LIN {X 0,Y 313.371,Z 298.457,A -85,B 0,C 180,E1 -15702.885,E2 -15702.885} C_VEL
LIN {X 0,Y 315.381,Z 300.73,A -85,B 0,C 180,E1 -15703.354,E2 -15703.354} C_VEL
LIN {X 0,Y 318.068,Z 304.811,A -85,B 0,C 180,E1 -15703.999,E2 -15703.999} C_VEL
LIN {X 0,Y 319.431,Z 306.632,A -85,B 0,C 180,E1 -15704.311,E2 -15704.311} C_VEL
LIN {X 0,Y 325.646,Z 315.457,A -85,B 0,C 180,E1 -15705.697,E2 -15705.697} C_VEL
LIN {X 0,Y 333.8,Z 327.772,A -85,B 0,C 180,E1 -15707.413,E2 -15707.413} C_VEL
LIN {X 0,Y 340.468,Z 338.749,A -85,B 0,C 180,E1 -15708.748,E2 -15708.748} C_VEL
LIN {X 0,Y 347.31,Z 351.998,A -85,B 0,C 180,E1 -15710.09,E2 -15710.09} C_VEL
LIN {X 0,Y 349.125,Z 355.68,A -85,B 0,C 180,E1 -15710.437,E2 -15710.437} C_VEL
LIN {X 0,Y 343.663,Z 493.802,A -85,B 0,C 180,E1 -15713.33,E2 -15713.33} C_VEL
LIN {X 0,Y 342.311,Z 510.914,A -85,B 0,C 180,E1 -15713.87,E2 -15713.87} C_VEL
LIN {X 0,Y 340.606,Z 527.054,A -85,B 0,C 180,E1 -15714.618,E2 -15714.618} C_VEL
LIN {X 0,Y 338.492,Z 542.365,A -85,B 0,C 180,E1 -15715.544,E2 -15715.544} C_VEL
LIN {X 0,Y 335.932,Z 557.671,A -85,B 0,C 180,E1 -15716.726,E2 -15716.726} C_VEL
LIN {X 0,Y 333.332,Z 571.386,A -85,B 0,C 180,E1 -15718.039,E2 -15718.039} C_VEL
LIN {X 0,Y 330.539,Z 584.215,A -85,B 0,C 180,E1 -15719.494,E2 -15719.494} C_VEL
LIN {X 0,Y 327.433,Z 597.477,A -85,B 0,C 180,E1 -15721.298,E2 -15721.298} C_VEL
LIN {X 0,Y 324.398,Z 609.578,A -85,B 0,C 180,E1 -15723.286,E2 -15723.286} C_VEL
LIN {X 0,Y 321.492,Z 620.685,A -85,B 0,C 180,E1 -15725.459,E2 -15725.459} C_VEL
LIN {X 0,Y 318.88,Z 630.612,A -85,B 0,C 180,E1 -15727.769,E2 -15727.769} C_VEL
LIN {X 0,Y 316.636,Z 639.434,A -85,B 0,C 180,E1 -15730.215,E2 -15730.215} C_VEL
LIN {X 0,Y 314.486,Z 647.965,A -85,B 0,C 180,E1 -15733.111,E2 -15733.111} C_VEL
LIN {X 0,Y 312.79,Z 655.524,A -85,B 0,C 180,E1 -15736.354,E2 -15736.354} C_VEL
LIN {X 0,Y 311.681,Z 661.259,A -85,B 0,C 180,E1 -15739.608,E2 -15739.608} C_VEL
LIN {X 0,Y 311.176,Z 664.614,A -85,B 0,C 180,E1 -15742.212,E2 -15742.212} C_VEL
LIN {X 0,Y 310.877,Z 667.053,A -85,B 0,C 180,E1 -15744.812,E2 -15744.812} C_VEL
LIN {X 0,Y 310.734,Z 668.437,A -85,B 0,C 180,E1 -15747.407,E2 -15747.407} C_VEL
LIN {X 0,Y 310.695,Z 668.97,A -85,B 0,C 180,E1 -15750,E2 -15750} C_VEL
LIN {X 0,Y 310.734,Z 668.477,A -85,B 0,C 180,E1 -15752.593,E2 -15752.593} C_VEL
LIN {X 0,Y 310.876,Z 667.132,A -85,B 0,C 180,E1 -15755.188,E2 -15755.188} C_VEL
LIN {X 0,Y 311.171,Z 664.734,A -85,B 0,C 180,E1 -15757.788,E2 -15757.788} C_VEL
LIN {X 0,Y 311.656,Z 661.427,A -85,B 0,C 180,E1 -15760.393,E2 -15760.393} C_VEL
LIN {X 0,Y 312.759,Z 655.741,A -85,B 0,C 180,E1 -15763.647,E2 -15763.647} C_VEL
LIN {X 0,Y 314.454,Z 648.254,A -85,B 0,C 180,E1 -15766.891,E2 -15766.891} C_VEL
LIN {X 0,Y 316.57,Z 639.766,A -85,B 0,C 180,E1 -15769.789,E2 -15769.789} C_VEL
LIN {X 0,Y 318.736,Z 631.273,A -85,B 0,C 180,E1 -15772.167,E2 -15772.167} C_VEL
LIN {X 0,Y 321.437,Z 621.161,A -85,B 0,C 180,E1 -15774.546,E2 -15774.546} C_VEL
LIN {X 0,Y 324.293,Z 610.151,A -85,B 0,C 180,E1 -15776.723,E2 -15776.723} C_VEL
LIN {X 0,Y 327.588,Z 597.113,A -85,B 0,C 180,E1 -15778.862,E2 -15778.862} C_VEL
LIN {X 0,Y 330.674,Z 583.796,A -85,B 0,C 180,E1 -15780.669,E2 -15780.669} C_VEL
LIN {X 0,Y 333.621,Z 570.298,A -85,B 0,C 180,E1 -15782.18,E2 -15782.18} C_VEL
LIN {X 0,Y 336.173,Z 556.682,A -85,B 0,C 180,E1 -15783.462,E2 -15783.462} C_VEL
LIN {X 0,Y 338.696,Z 541.625,A -85,B 0,C 180,E1 -15784.613,E2 -15784.613} C_VEL
LIN {X 0,Y 339.449,Z 536.57,A -85,B 0,C 180,E1 -15784.931,E2 -15784.931} C_VEL
LIN {X 0,Y 339.734,Z 531.151,A -85,B 0,C 180,E1 -15785.32,E2 -15785.32} C_VEL
LIN {X 0,Y 337.206,Z 513.489,A -85,B 0,C 180,E1 -15786.764,E2 -15786.764} C_VEL
LIN {X 0,Y 337.05,Z 507.877,A -85,B 0,C 180,E1 -15787.068,E2 -15787.068} C_VEL
LIN {X 0,Y 338.19,Z 491.988,A -85,B 0,C 180,E1 -15787.544,E2 -15787.544} C_VEL
LIN {X 0,Y 343.655,Z 358.179,A -85,B 0,C 180,E1 -15790.378,E2 -15790.378} C_VEL
LIN {X 0,Y 336.006,Z 343.116,A -85,B 0,C 180,E1 -15791.927,E2 -15791.927} C_VEL
LIN {X 0,Y 327.751,Z 329.585,A -85,B 0,C 180,E1 -15793.647,E2 -15793.647} C_VEL
LIN {X 0,Y 317.849,Z 314.862,A -85,B 0,C 180,E1 -15795.853,E2 -15795.853} C_VEL
LIN {X 0,Y 312.292,Z 307.072,A -85,B 0,C 180,E1 -15797.179,E2 -15797.179} C_VEL
LIN {X 0,Y 309.294,Z 303.031,A -85,B 0,C 180,E1 -15797.923,E2 -15797.923} C_VEL
LIN {X 0,Y 308.538,Z 301.775,A -85,B 0,C 180,E1 -15798.123,E2 -15798.123} C_VEL
LIN {X 0,Y 306.51,Z 299.73,A -85,B 0,C 180,E1 -15798.621,E2 -15798.621} C_VEL
LIN {X 0,Y 305.504,Z 297.232,A -85,B 0,C 180,E1 -15798.925,E2 -15798.925} C_VEL
LIN {X 0,Y 305.437,Z 296.736,A -85,B 0,C 180,E1 -15798.999,E2 -15798.999} C_VEL
LIN {X 0,Y 305.474,Z 296.741,A -85,B 0,C 180,E1 -15801.597,E2 -15801.597} C_VEL
LIN {X 0,Y 305.461,Z 296.748,A -85,B 0,C 180,E1 -15804.886,E2 -15804.886} C_VEL
LIN {X 0,Y 305.448,Z 296.735,A -85,B 0,C 180,E1 -15808.355,E2 -15808.355} C_VEL
LIN {X 0,Y 305.511,Z 296.727,A -85,B 0,C 180,E1 -15811.113,E2 -15811.113} C_VEL
LIN {X 0,Y 305.569,Z 296.727,A -85,B 0,C 180,E1 -15814.088,E2 -15814.088} C_VEL
LIN {X 0,Y 305.498,Z 296.717,A -85,B 0,C 180,E1 -15818.403,E2 -15818.403} C_VEL
LIN {X 0,Y 305.588,Z 296.732,A -85,B 0,C 180,E1 -15821.217,E2 -15821.217} C_VEL
LIN {X 0,Y 305.647,Z 296.704,A -85,B 0,C 180,E1 -15825.349,E2 -15825.349} C_VEL
LIN {X 0,Y 305.636,Z 296.7,A -85,B 0,C 180,E1 -15829.399,E2 -15829.399} C_VEL
LIN {X 0,Y 305.811,Z 296.687,A -85,B 0,C 180,E1 -15832.074,E2 -15832.074} C_VEL
LIN {X 0,Y 305.687,Z 296.715,A -85,B 0,C 180,E1 -15834.723,E2 -15834.723} C_VEL
LIN {X 0,Y 305.955,Z 296.666,A -85,B 0,C 180,E1 -15838.684,E2 -15838.684} C_VEL
LIN {X 0,Y 305.955,Z 296.683,A -85,B 0,C 180,E1 -15841.316,E2 -15841.316} C_VEL
LIN {X 0,Y 305.85,Z 296.696,A -85,B 0,C 180,E1 -15846.597,E2 -15846.597} C_VEL
LIN {X 0,Y 305.734,Z 296.693,A -85,B 0,C 180,E1 -15849.26,E2 -15849.26} C_VEL
LIN {X 0,Y 305.587,Z 296.732,A -85,B 0,C 180,E1 -15853.296,E2 -15853.296} C_VEL
LIN {X 0,Y 305.592,Z 296.729,A -85,B 0,C 180,E1 -15856.02,E2 -15856.02} C_VEL
LIN {X 0,Y 305.575,Z 296.736,A -85,B 0,C 180,E1 -15859.445,E2 -15859.445} C_VEL
LIN {X 0,Y 305.488,Z 296.749,A -85,B 0,C 180,E1 -15863.041,E2 -15863.041} C_VEL
LIN {X 0,Y 305.545,Z 296.743,A -85,B 0,C 180,E1 -15866.227,E2 -15866.227} C_VEL
LIN {X 0,Y 305.494,Z 296.749,A -85,B 0,C 180,E1 -15869.05,E2 -15869.05} C_VEL
LIN {X 0,Y 305.442,Z 296.757,A -85,B 0,C 180,E1 -15871.952,E2 -15871.952} C_VEL
LIN {X 0,Y 305.46,Z 296.75,A -85,B 0,C 180,E1 -15875.113,E2 -15875.113} C_VEL
LIN {X 0,Y 305.447,Z 296.757,A -85,B 0,C 180,E1 -15878.529,E2 -15878.529} C_VEL
LIN {X 0,Y 305.465,Z 296.923,A -85,B 0,C 180,E1 -15879.468,E2 -15879.468} C_VEL
LIN {X 0,Y 308.218,Z 303.518,A -85,B 0,C 180,E1 -15881.505,E2 -15881.505} C_VEL
LIN {X 0,Y 316.88,Z 316.875,A -85,B 0,C 180,E1 -15883.664,E2 -15883.664} C_VEL
LIN {X 0,Y 324.584,Z 329.236,A -85,B 0,C 180,E1 -15885.438,E2 -15885.438} C_VEL
LIN {X 0,Y 332.597,Z 343.649,A -85,B 0,C 180,E1 -15887.189,E2 -15887.189} C_VEL
LIN {X 0,Y 340.914,Z 360.154,A -85,B 0,C 180,E1 -15888.915,E2 -15888.915} C_VEL
LIN {X 0,Y 343.483,Z 365.809,A -85,B 0,C 180,E1 -15889.437,E2 -15889.437} C_VEL
LIN {X 0,Y 337.406,Z 512.132,A -85,B 0,C 180,E1 -15892.54,E2 -15892.54} C_VEL
LIN {X 0,Y 335.817,Z 529.145,A -85,B 0,C 180,E1 -15893.104,E2 -15893.104} C_VEL
LIN {X 0,Y 333.935,Z 544.026,A -85,B 0,C 180,E1 -15893.801,E2 -15893.801} C_VEL
LIN {X 0,Y 331.666,Z 559.189,A -85,B 0,C 180,E1 -15894.731,E2 -15894.731} C_VEL
LIN {X 0,Y 328.916,Z 574.15,A -85,B 0,C 180,E1 -15895.883,E2 -15895.883} C_VEL
LIN {X 0,Y 325.719,Z 589.41,A -85,B 0,C 180,E1 -15897.356,E2 -15897.356} C_VEL
LIN {X 0,Y 322.401,Z 603.395,A -85,B 0,C 180,E1 -15899.003,E2 -15899.003} C_VEL
LIN {X 0,Y 319.483,Z 615.351,A -85,B 0,C 180,E1 -15900.696,E2 -15900.696} C_VEL
LIN {X 0,Y 316.666,Z 626.009,A -85,B 0,C 180,E1 -15902.465,E2 -15902.465} C_VEL
LIN {X 0,Y 313.934,Z 636.294,A -85,B 0,C 180,E1 -15904.473,E2 -15904.473} C_VEL
LIN {X 0,Y 311.298,Z 646.17,A -85,B 0,C 180,E1 -15906.729,E2 -15906.729} C_VEL
LIN {X 0,Y 308.826,Z 655.677,A -85,B 0,C 180,E1 -15909.345,E2 -15909.345} C_VEL
LIN {X 0,Y 306.925,Z 663.639,A -85,B 0,C 180,E1 -15911.994,E2 -15911.994} C_VEL
LIN {X 0,Y 305.507,Z 670.29,A -85,B 0,C 180,E1 -15914.661,E2 -15914.661} C_VEL
LIN {X 0,Y 304.548,Z 675.693,A -85,B 0,C 180,E1 -15917.336,E2 -15917.336} C_VEL
LIN {X 0,Y 304.001,Z 679.031,A -85,B 0,C 180,E1 -15919.342,E2 -15919.342} C_VEL
LIN {X 0,Y 303.684,Z 682.467,A -85,B 0,C 180,E1 -15922.019,E2 -15922.019} C_VEL
LIN {X 0,Y 303.595,Z 684.967,A -85,B 0,C 180,E1 -15924.687,E2 -15924.687} C_VEL
LIN {X 0,Y 303.594,Z 686.378,A -85,B 0,C 180,E1 -15927.346,E2 -15927.346} C_VEL
LIN {X 0,Y 303.601,Z 686.908,A -85,B 0,C 180,E1 -15930,E2 -15930} C_VEL
LIN {X 0,Y 303.594,Z 686.371,A -85,B 0,C 180,E1 -15932.654,E2 -15932.654} C_VEL
LIN {X 0,Y 303.623,Z 684.76,A -85,B 0,C 180,E1 -15935.545,E2 -15935.545} C_VEL
LIN {X 0,Y 303.684,Z 682.446,A -85,B 0,C 180,E1 -15937.982,E2 -15937.982} C_VEL
LIN {X 0,Y 304.001,Z 679.004,A -85,B 0,C 180,E1 -15940.658,E2 -15940.658} C_VEL
LIN {X 0,Y 305.004,Z 673.131,A -85,B 0,C 180,E1 -15944.001,E2 -15944.001} C_VEL
LIN {X 0,Y 306.516,Z 665.413,A -85,B 0,C 180,E1 -15947.342,E2 -15947.342} C_VEL
LIN {X 0,Y 308.603,Z 656.719,A -85,B 0,C 180,E1 -15950.322,E2 -15950.322} C_VEL
LIN {X 0,Y 310.955,Z 647.339,A -85,B 0,C 180,E1 -15952.946,E2 -15952.946} C_VEL
LIN {X 0,Y 313.537,Z 637.697,A -85,B 0,C 180,E1 -15955.207,E2 -15955.207} C_VEL
LIN {X 0,Y 316.215,Z 627.523,A -85,B 0,C 180,E1 -15957.251,E2 -15957.251} C_VEL
LIN {X 0,Y 319.449,Z 615.221,A -85,B 0,C 180,E1 -15959.308,E2 -15959.308} C_VEL
LIN {X 0,Y 322.649,Z 602.059,A -85,B 0,C 180,E1 -15961.153,E2 -15961.153} C_VEL
LIN {X 0,Y 325.761,Z 588.634,A -85,B 0,C 180,E1 -15962.713,E2 -15962.713} C_VEL
LIN {X 0,Y 328.889,Z 573.901,A -85,B 0,C 180,E1 -15964.12,E2 -15964.12} C_VEL
LIN {X 0,Y 331.819,Z 557.903,A -85,B 0,C 180,E1 -15965.344,E2 -15965.344} C_VEL
LIN {X 0,Y 334.109,Z 542.363,A -85,B 0,C 180,E1 -15966.271,E2 -15966.271} C_VEL
LIN {X 0,Y 336.028,Z 526.804,A -85,B 0,C 180,E1 -15966.963,E2 -15966.963} C_VEL
LIN {X 0,Y 337.482,Z 510.229,A -85,B 0,C 180,E1 -15967.484,E2 -15967.484} C_VEL
LIN {X 0,Y 343.385,Z 365.697,A -85,B 0,C 180,E1 -15970.551,E2 -15970.551} C_VEL
LIN {X 0,Y 335.117,Z 348.583,A -85,B 0,C 180,E1 -15972.244,E2 -15972.244} C_VEL
LIN {X 0,Y 326.72,Z 332.985,A -85,B 0,C 180,E1 -15974.048,E2 -15974.048} C_VEL
LIN {X 0,Y 318.181,Z 318.811,A -85,B 0,C 180,E1 -15975.99,E2 -15975.99} C_VEL
LIN {X 0,Y 313.283,Z 311.23,A -85,B 0,C 180,E1 -15977.167,E2 -15977.167} C_VEL
LIN {X 0,Y 308.364,Z 303.718,A -85,B 0,C 180,E1 -15978.411,E2 -15978.411} C_VEL
LIN {X 0,Y 307.25,Z 301.662,A -85,B 0,C 180,E1 -15979.011,E2 -15979.011} C_VEL
LIN {X 0,Y 305.448,Z 296.74,A -85,B 0,C 180,E1 -15980.583,E2 -15980.583} C_VEL
LIN {X 0,Y 305.479,Z 296.742,A -85,B 0,C 180,E1 -15983.632,E2 -15983.632} C_VEL
LIN {X 0,Y 305.463,Z 296.745,A -85,B 0,C 180,E1 -15986.483,E2 -15986.483} C_VEL
LIN {X 0,Y 305.461,Z 296.742,A -85,B 0,C 180,E1 -15989.591,E2 -15989.591} C_VEL
LIN {X 0,Y 305.519,Z 296.735,A -85,B 0,C 180,E1 -15992.609,E2 -15992.609} C_VEL
LIN {X 0,Y 305.506,Z 296.737,A -85,B 0,C 180,E1 -15995.539,E2 -15995.539} C_VEL
LIN {X 0,Y 305.517,Z 296.709,A -85,B 0,C 180,E1 -15999.815,E2 -15999.815} C_VEL
LIN {X 0,Y 305.573,Z 296.732,A -85,B 0,C 180,E1 -16002.603,E2 -16002.603} C_VEL
LIN {X 0,Y 305.647,Z 296.697,A -85,B 0,C 180,E1 -16005.349,E2 -16005.349} C_VEL
LIN {X 0,Y 305.634,Z 296.725,A -85,B 0,C 180,E1 -16009.4,E2 -16009.4} C_VEL
LIN {X 0,Y 305.795,Z 296.681,A -85,B 0,C 180,E1 -16012.074,E2 -16012.074} C_VEL
LIN {X 0,Y 305.685,Z 296.69,A -85,B 0,C 180,E1 -16014.724,E2 -16014.724} C_VEL
LIN {X 0,Y 305.954,Z 296.672,A -85,B 0,C 180,E1 -16018.684,E2 -16018.684} C_VEL
LIN {X 0,Y 305.954,Z 296.649,A -85,B 0,C 180,E1 -16021.316,E2 -16021.316} C_VEL
LIN {X 0,Y 305.686,Z 296.716,A -85,B 0,C 180,E1 -16025.277,E2 -16025.277} C_VEL
LIN {X 0,Y 305.795,Z 296.667,A -85,B 0,C 180,E1 -16027.926,E2 -16027.926} C_VEL
LIN {X 0,Y 305.602,Z 296.73,A -85,B 0,C 180,E1 -16031.945,E2 -16031.945} C_VEL
LIN {X 0,Y 305.636,Z 296.691,A -85,B 0,C 180,E1 -16035.035,E2 -16035.035} C_VEL
LIN {X 0,Y 305.574,Z 296.73,A -85,B 0,C 180,E1 -16039.444,E2 -16039.444} C_VEL
LIN {X 0,Y 305.485,Z 296.72,A -85,B 0,C 180,E1 -16043.04,E2 -16043.04} C_VEL
LIN {X 0,Y 305.53,Z 296.726,A -85,B 0,C 180,E1 -16046.221,E2 -16046.221} C_VEL
LIN {X 0,Y 305.493,Z 296.723,A -85,B 0,C 180,E1 -16049.05,E2 -16049.05} C_VEL
LIN {X 0,Y 305.443,Z 296.744,A -85,B 0,C 180,E1 -16051.952,E2 -16051.952} C_VEL
LIN {X 0,Y 305.461,Z 296.743,A -85,B 0,C 180,E1 -16055.113,E2 -16055.113} C_VEL
LIN {X 0,Y 305.439,Z 296.727,A -85,B 0,C 180,E1 -16058.527,E2 -16058.527} C_VEL
LIN {X 0,Y 305.428,Z 296.738,A -85,B 0,C 180,E1 -16061.172,E2 -16061.172} C_VEL
LIN {X 0,Y 306.387,Z 299.529,A -85,B 0,C 180,E1 -16061.485,E2 -16061.485} C_VEL
LIN {X 0,Y 308.565,Z 301.776,A -85,B 0,C 180,E1 -16062.021,E2 -16062.021} C_VEL
LIN {X 0,Y 311.419,Z 305.968,A -85,B 0,C 180,E1 -16062.745,E2 -16062.745} C_VEL
LIN {X 0,Y 312.907,Z 308.125,A -85,B 0,C 180,E1 -16063.113,E2 -16063.113} C_VEL
LIN {X 0,Y 316.163,Z 312.626,A -85,B 0,C 180,E1 -16063.89,E2 -16063.89} C_VEL
LIN {X 0,Y 324.196,Z 324.178,A -85,B 0,C 180,E1 -16065.71,E2 -16065.71} C_VEL
LIN {X 0,Y 334.002,Z 339.669,A -85,B 0,C 180,E1 -16067.786,E2 -16067.786} C_VEL
LIN {X 0,Y 341.105,Z 353.04,A -85,B 0,C 180,E1 -16069.234,E2 -16069.234} C_VEL
LIN {X 0,Y 343.559,Z 358.14,A -85,B 0,C 180,E1 -16069.726,E2 -16069.726} C_VEL
LIN {X 0,Y 337.994,Z 494.396,A -85,B 0,C 180,E1 -16072.623,E2 -16072.623} C_VEL
LIN {X 0,Y 336.62,Z 511.134,A -85,B 0,C 180,E1 -16073.159,E2 -16073.159} C_VEL
LIN {X 0,Y 334.856,Z 527.27,A -85,B 0,C 180,E1 -16073.916,E2 -16073.916} C_VEL
LIN {X 0,Y 332.677,Z 542.578,A -85,B 0,C 180,E1 -16074.854,E2 -16074.854} C_VEL
LIN {X 0,Y 330.074,Z 557.53,A -85,B 0,C 180,E1 -16076.019,E2 -16076.019} C_VEL
LIN {X 0,Y 327.295,Z 571.663,A -85,B 0,C 180,E1 -16077.386,E2 -16077.386} C_VEL
LIN {X 0,Y 324.157,Z 585.594,A -85,B 0,C 180,E1 -16079.008,E2 -16079.008} C_VEL
LIN {X 0,Y 320.921,Z 598.663,A -85,B 0,C 180,E1 -16080.839,E2 -16080.839} C_VEL
LIN {X 0,Y 318.032,Z 609.79,A -85,B 0,C 180,E1 -16082.707,E2 -16082.707} C_VEL
LIN {X 0,Y 315.008,Z 620.896,A -85,B 0,C 180,E1 -16084.919,E2 -16084.919} C_VEL
LIN {X 0,Y 312.133,Z 631.279,A -85,B 0,C 180,E1 -16087.392,E2 -16087.392} C_VEL
LIN {X 0,Y 309.897,Z 639.645,A -85,B 0,C 180,E1 -16089.767,E2 -16089.767} C_VEL
LIN {X 0,Y 307.634,Z 648.176,A -85,B 0,C 180,E1 -16092.723,E2 -16092.723} C_VEL
LIN {X 0,Y 306.113,Z 654.329,A -85,B 0,C 180,E1 -16095.372,E2 -16095.372} C_VEL
LIN {X 0,Y 304.988,Z 659.369,A -85,B 0,C 180,E1 -16098.03,E2 -16098.03} C_VEL
LIN {X 0,Y 304.357,Z 663.262,A -85,B 0,C 180,E1 -16100.698,E2 -16100.698} C_VEL
LIN {X 0,Y 303.843,Z 666.728,A -85,B 0,C 180,E1 -16104.047,E2 -16104.047} C_VEL
LIN {X 0,Y 303.733,Z 668.058,A -85,B 0,C 180,E1 -16106.02,E2 -16106.02} C_VEL
LIN {X 0,Y 303.605,Z 669.022,A -85,B 0,C 180,E1 -16108.674,E2 -16108.674} C_VEL
LIN {X 0,Y 303.604,Z 669.035,A -85,B 0,C 180,E1 -16111.326,E2 -16111.326} C_VEL
LIN {X 0,Y 303.733,Z 668.124,A -85,B 0,C 180,E1 -16113.98,E2 -16113.98} C_VEL
LIN {X 0,Y 303.939,Z 666.25,A -85,B 0,C 180,E1 -16116.639,E2 -16116.639} C_VEL
LIN {X 0,Y 304.335,Z 663.406,A -85,B 0,C 180,E1 -16119.303,E2 -16119.303} C_VEL
LIN {X 0,Y 304.972,Z 659.537,A -85,B 0,C 180,E1 -16121.97,E2 -16121.97} C_VEL
LIN {X 0,Y 306.078,Z 654.556,A -85,B 0,C 180,E1 -16124.63,E2 -16124.63} C_VEL
LIN {X 0,Y 307.605,Z 648.462,A -85,B 0,C 180,E1 -16127.278,E2 -16127.278} C_VEL
LIN {X 0,Y 309.849,Z 639.973,A -85,B 0,C 180,E1 -16130.237,E2 -16130.237} C_VEL
LIN {X 0,Y 312.262,Z 630.931,A -85,B 0,C 180,E1 -16132.81,E2 -16132.81} C_VEL
LIN {X 0,Y 314.945,Z 621.367,A -85,B 0,C 180,E1 -16135.086,E2 -16135.086} C_VEL
LIN {X 0,Y 317.917,Z 610.357,A -85,B 0,C 180,E1 -16137.303,E2 -16137.303} C_VEL
LIN {X 0,Y 321.357,Z 597.318,A -85,B 0,C 180,E1 -16139.476,E2 -16139.476} C_VEL
LIN {X 0,Y 324.552,Z 584,A -85,B 0,C 180,E1 -16141.312,E2 -16141.312} C_VEL
LIN {X 0,Y 327.368,Z 571.714,A -85,B 0,C 180,E1 -16142.715,E2 -16142.715} C_VEL
LIN {X 0,Y 329.943,Z 558.64,A -85,B 0,C 180,E1 -16143.996,E2 -16143.996} C_VEL
LIN {X 0,Y 332.685,Z 542.837,A -85,B 0,C 180,E1 -16145.238,E2 -16145.238} C_VEL
LIN {X 0,Y 334.892,Z 527.592,A -85,B 0,C 180,E1 -16146.173,E2 -16146.173} C_VEL
LIN {X 0,Y 336.557,Z 512.495,A -85,B 0,C 180,E1 -16146.895,E2 -16146.895} C_VEL
LIN {X 0,Y 337.05,Z 507.877,A -85,B 0,C 180,E1 -16147.068,E2 -16147.068} C_VEL
LIN {X 0,Y 336.904,Z 502.194,A -85,B 0,C 180,E1 -16147.353,E2 -16147.353} C_VEL
LIN {X 0,Y 333.672,Z 485.599,A -85,B 0,C 180,E1 -16148.34,E2 -16148.34} C_VEL
LIN {X 0,Y 333.176,Z 479.864,A -85,B 0,C 180,E1 -16148.563,E2 -16148.563} C_VEL
LIN {X 0,Y 333.222,Z 477.917,A -85,B 0,C 180,E1 -16148.609,E2 -16148.609} C_VEL
LIN {X 0,Y 338.151,Z 360.596,A -85,B 0,C 180,E1 -16151.114,E2 -16151.114} C_VEL
LIN {X 0,Y 330.874,Z 346.293,A -85,B 0,C 180,E1 -16152.643,E2 -16152.643} C_VEL
LIN {X 0,Y 321.604,Z 331.27,A -85,B 0,C 180,E1 -16154.655,E2 -16154.655} C_VEL
LIN {X 0,Y 313.397,Z 319.25,A -85,B 0,C 180,E1 -16156.56,E2 -16156.56} C_VEL
LIN {X 0,Y 307.865,Z 311.387,A -85,B 0,C 180,E1 -16157.933,E2 -16157.933} C_VEL
LIN {X 0,Y 304.735,Z 307.162,A -85,B 0,C 180,E1 -16158.742,E2 -16158.742} C_VEL
LIN {X 0,Y 302.436,Z 304.111,A -85,B 0,C 180,E1 -16159.353,E2 -16159.353} C_VEL
LIN {X 0,Y 301.523,Z 302.649,A -85,B 0,C 180,E1 -16159.61,E2 -16159.61} C_VEL
LIN {X 0,Y 299.387,Z 300.453,A -85,B 0,C 180,E1 -16160.177,E2 -16160.177} C_VEL
LIN {X 0,Y 298.482,Z 298.213,A -85,B 0,C 180,E1 -16160.47,E2 -16160.47} C_VEL
LIN {X 0,Y 298.395,Z 297.625,A -85,B 0,C 180,E1 -16160.55,E2 -16160.55} C_VEL
LIN {X 0,Y 298.417,Z 297.613,A -85,B 0,C 180,E1 -16163.93,E2 -16163.93} C_VEL
LIN {X 0,Y 298.392,Z 297.61,A -85,B 0,C 180,E1 -16167.984,E2 -16167.984} C_VEL
LIN {X 0,Y 298.457,Z 297.597,A -85,B 0,C 180,E1 -16171.903,E2 -16171.903} C_VEL
LIN {X 0,Y 298.484,Z 297.618,A -85,B 0,C 180,E1 -16174.924,E2 -16174.924} C_VEL
LIN {X 0,Y 298.448,Z 297.604,A -85,B 0,C 180,E1 -16179.315,E2 -16179.315} C_VEL
LIN {X 0,Y 298.535,Z 297.597,A -85,B 0,C 180,E1 -16182.179,E2 -16182.179} C_VEL
LIN {X 0,Y 298.591,Z 297.577,A -85,B 0,C 180,E1 -16184.994,E2 -16184.994} C_VEL
LIN {X 0,Y 298.591,Z 297.58,A -85,B 0,C 180,E1 -16189.146,E2 -16189.146} C_VEL
LIN {X 0,Y 298.756,Z 297.561,A -85,B 0,C 180,E1 -16191.886,E2 -16191.886} C_VEL
LIN {X 0,Y 298.658,Z 297.592,A -85,B 0,C 180,E1 -16194.599,E2 -16194.599} C_VEL
LIN {X 0,Y 298.921,Z 297.541,A -85,B 0,C 180,E1 -16198.653,E2 -16198.653} C_VEL
LIN {X 0,Y 298.922,Z 297.559,A -85,B 0,C 180,E1 -16201.347,E2 -16201.347} C_VEL
LIN {X 0,Y 298.796,Z 297.576,A -85,B 0,C 180,E1 -16206.754,E2 -16206.754} C_VEL
LIN {X 0,Y 298.678,Z 297.568,A -85,B 0,C 180,E1 -16209.48,E2 -16209.48} C_VEL
LIN {X 0,Y 298.55,Z 297.61,A -85,B 0,C 180,E1 -16213.615,E2 -16213.615} C_VEL
LIN {X 0,Y 298.547,Z 297.608,A -85,B 0,C 180,E1 -16216.409,E2 -16216.409} C_VEL
LIN {X 0,Y 298.509,Z 297.616,A -85,B 0,C 180,E1 -16219.655,E2 -16219.655} C_VEL
LIN {X 0,Y 298.455,Z 297.622,A -85,B 0,C 180,E1 -16223.598,E2 -16223.598} C_VEL
LIN {X 0,Y 298.487,Z 297.619,A -85,B 0,C 180,E1 -16226.574,E2 -16226.574} C_VEL
LIN {X 0,Y 298.418,Z 297.626,A -85,B 0,C 180,E1 -16229.641,E2 -16229.641} C_VEL
LIN {X 0,Y 298.393,Z 297.629,A -85,B 0,C 180,E1 -16232.8,E2 -16232.8} C_VEL
LIN {X 0,Y 298.444,Z 297.63,A -85,B 0,C 180,E1 -16236.808,E2 -16236.808} C_VEL
LIN {X 0,Y 298.451,Z 297.815,A -85,B 0,C 180,E1 -16238.102,E2 -16238.102} C_VEL
LIN {X 0,Y 300.626,Z 303.24,A -85,B 0,C 180,E1 -16239.843,E2 -16239.843} C_VEL
LIN {X 0,Y 305.32,Z 310.055,A -85,B 0,C 180,E1 -16241.119,E2 -16241.119} C_VEL
LIN {X 0,Y 312.367,Z 320.859,A -85,B 0,C 180,E1 -16242.927,E2 -16242.927} C_VEL
LIN {X 0,Y 319.198,Z 331.957,A -85,B 0,C 180,E1 -16244.569,E2 -16244.569} C_VEL
LIN {X 0,Y 325.524,Z 343.068,A -85,B 0,C 180,E1 -16246.015,E2 -16246.015} C_VEL
LIN {X 0,Y 335.297,Z 362.201,A -85,B 0,C 180,E1 -16248.136,E2 -16248.136} C_VEL
LIN {X 0,Y 337.953,Z 368.075,A -85,B 0,C 180,E1 -16248.698,E2 -16248.698} C_VEL
LIN {X 0,Y 334.71,Z 443.669,A -85,B 0,C 180,E1 -16250.303,E2 -16250.303} C_VEL
LIN {X 0,Y 331.78,Z 512.373,A -85,B 0,C 180,E1 -16251.807,E2 -16251.807} C_VEL
LIN {X 0,Y 330.063,Z 529.866,A -85,B 0,C 180,E1 -16252.398,E2 -16252.398} C_VEL
LIN {X 0,Y 328.026,Z 545.129,A -85,B 0,C 180,E1 -16253.137,E2 -16253.137} C_VEL
LIN {X 0,Y 325.858,Z 558.986,A -85,B 0,C 180,E1 -16254.005,E2 -16254.005} C_VEL
LIN {X 0,Y 323.025,Z 573.947,A -85,B 0,C 180,E1 -16255.172,E2 -16255.172} C_VEL
LIN {X 0,Y 319.675,Z 589.204,A -85,B 0,C 180,E1 -16256.659,E2 -16256.659} C_VEL
LIN {X 0,Y 316.3,Z 603.19,A -85,B 0,C 180,E1 -16258.337,E2 -16258.337} C_VEL
LIN {X 0,Y 313.247,Z 615.144,A -85,B 0,C 180,E1 -16260.053,E2 -16260.053} C_VEL
LIN {X 0,Y 310.02,Z 626.87,A -85,B 0,C 180,E1 -16262.042,E2 -16262.042} C_VEL
LIN {X 0,Y 306.601,Z 639.077,A -85,B 0,C 180,E1 -16264.546,E2 -16264.546} C_VEL
LIN {X 0,Y 303.993,Z 648.448,A -85,B 0,C 180,E1 -16266.858,E2 -16266.858} C_VEL
LIN {X 0,Y 301.541,Z 657.589,A -85,B 0,C 180,E1 -16269.537,E2 -16269.537} C_VEL
LIN {X 0,Y 299.633,Z 665.256,A -85,B 0,C 180,E1 -16272.247,E2 -16272.247} C_VEL
LIN {X 0,Y 298.021,Z 673.034,A -85,B 0,C 180,E1 -16275.703,E2 -16275.703} C_VEL
LIN {X 0,Y 296.954,Z 678.822,A -85,B 0,C 180,E1 -16279.086,E2 -16279.086} C_VEL
LIN {X 0,Y 296.594,Z 682.258,A -85,B 0,C 180,E1 -16281.826,E2 -16281.826} C_VEL
LIN {X 0,Y 296.51,Z 684.759,A -85,B 0,C 180,E1 -16284.56,E2 -16284.56} C_VEL
LIN {X 0,Y 296.52,Z 686.172,A -85,B 0,C 180,E1 -16287.283,E2 -16287.283} C_VEL
LIN {X 0,Y 296.516,Z 686.701,A -85,B 0,C 180,E1 -16290,E2 -16290} C_VEL
LIN {X 0,Y 296.52,Z 686.164,A -85,B 0,C 180,E1 -16292.717,E2 -16292.717} C_VEL
LIN {X 0,Y 296.51,Z 684.744,A -85,B 0,C 180,E1 -16295.44,E2 -16295.44} C_VEL
LIN {X 0,Y 296.594,Z 682.236,A -85,B 0,C 180,E1 -16298.174,E2 -16298.174} C_VEL
LIN {X 0,Y 296.954,Z 678.794,A -85,B 0,C 180,E1 -16300.914,E2 -16300.914} C_VEL
LIN {X 0,Y 298.006,Z 672.993,A -85,B 0,C 180,E1 -16304.299,E2 -16304.299} C_VEL
LIN {X 0,Y 299.633,Z 665.201,A -85,B 0,C 180,E1 -16307.753,E2 -16307.753} C_VEL
LIN {X 0,Y 301.821,Z 656.558,A -85,B 0,C 180,E1 -16310.782,E2 -16310.782} C_VEL
LIN {X 0,Y 304.322,Z 647.126,A -85,B 0,C 180,E1 -16313.476,E2 -16313.476} C_VEL
LIN {X 0,Y 307.048,Z 637.485,A -85,B 0,C 180,E1 -16315.778,E2 -16315.778} C_VEL
LIN {X 0,Y 309.929,Z 626.956,A -85,B 0,C 180,E1 -16317.925,E2 -16317.925} C_VEL
LIN {X 0,Y 313.379,Z 614.024,A -85,B 0,C 180,E1 -16320.119,E2 -16320.119} C_VEL
LIN {X 0,Y 316.828,Z 600.667,A -85,B 0,C 180,E1 -16321.978,E2 -16321.978} C_VEL
LIN {X 0,Y 319.979,Z 587.569,A -85,B 0,C 180,E1 -16323.493,E2 -16323.493} C_VEL
LIN {X 0,Y 322.987,Z 573.687,A -85,B 0,C 180,E1 -16324.832,E2 -16324.832} C_VEL
LIN {X 0,Y 326.02,Z 557.689,A -85,B 0,C 180,E1 -16326.07,E2 -16326.07} C_VEL
LIN {X 0,Y 328.391,Z 542.148,A -85,B 0,C 180,E1 -16327.007,E2 -16327.007} C_VEL
LIN {X 0,Y 330.374,Z 526.585,A -85,B 0,C 180,E1 -16327.705,E2 -16327.705} C_VEL
LIN {X 0,Y 331.871,Z 510.004,A -85,B 0,C 180,E1 -16328.23,E2 -16328.23} C_VEL
LIN {X 0,Y 337.871,Z 367.992,A -85,B 0,C 180,E1 -16331.286,E2 -16331.286} C_VEL
LIN {X 0,Y 329.812,Z 351.348,A -85,B 0,C 180,E1 -16332.999,E2 -16332.999} C_VEL
LIN {X 0,Y 322.222,Z 337.197,A -85,B 0,C 180,E1 -16334.692,E2 -16334.692} C_VEL
LIN {X 0,Y 314.16,Z 323.656,A -85,B 0,C 180,E1 -16336.591,E2 -16336.591} C_VEL
LIN {X 0,Y 307.71,Z 313.601,A -85,B 0,C 180,E1 -16338.208,E2 -16338.208} C_VEL
LIN {X 0,Y 303.879,Z 307.934,A -85,B 0,C 180,E1 -16339.216,E2 -16339.216} C_VEL
LIN {X 0,Y 300.399,Z 302.877,A -85,B 0,C 180,E1 -16340.176,E2 -16340.176} C_VEL
LIN {X 0,Y 299.837,Z 301.043,A -85,B 0,C 180,E1 -16340.739,E2 -16340.739} C_VEL
LIN {X 0,Y 298.562,Z 298.272,A -85,B 0,C 180,E1 -16341.704,E2 -16341.704} C_VEL
LIN {X 0,Y 298.433,Z 297.616,A -85,B 0,C 180,E1 -16341.965,E2 -16341.965} C_VEL
LIN {X 0,Y 298.406,Z 297.62,A -85,B 0,C 180,E1 -16345.581,E2 -16345.581} C_VEL
LIN {X 0,Y 298.394,Z 297.628,A -85,B 0,C 180,E1 -16348.791,E2 -16348.791} C_VEL
LIN {X 0,Y 298.461,Z 297.618,A -85,B 0,C 180,E1 -16351.904,E2 -16351.904} C_VEL
LIN {X 0,Y 298.484,Z 297.614,A -85,B 0,C 180,E1 -16354.924,E2 -16354.924} C_VEL
LIN {X 0,Y 298.448,Z 297.591,A -85,B 0,C 180,E1 -16359.315,E2 -16359.315} C_VEL
LIN {X 0,Y 298.536,Z 297.603,A -85,B 0,C 180,E1 -16362.18,E2 -16362.18} C_VEL
LIN {X 0,Y 298.591,Z 297.58,A -85,B 0,C 180,E1 -16364.995,E2 -16364.995} C_VEL
LIN {X 0,Y 298.59,Z 297.599,A -85,B 0,C 180,E1 -16369.147,E2 -16369.147} C_VEL
LIN {X 0,Y 298.739,Z 297.562,A -85,B 0,C 180,E1 -16371.886,E2 -16371.886} C_VEL
LIN {X 0,Y 298.656,Z 297.563,A -85,B 0,C 180,E1 -16374.599,E2 -16374.599} C_VEL
LIN {X 0,Y 298.921,Z 297.548,A -85,B 0,C 180,E1 -16378.653,E2 -16378.653} C_VEL
LIN {X 0,Y 298.92,Z 297.524,A -85,B 0,C 180,E1 -16381.347,E2 -16381.347} C_VEL
LIN {X 0,Y 298.786,Z 297.55,A -85,B 0,C 180,E1 -16386.754,E2 -16386.754} C_VEL
LIN {X 0,Y 298.634,Z 297.567,A -85,B 0,C 180,E1 -16389.482,E2 -16389.482} C_VEL
LIN {X 0,Y 298.551,Z 297.587,A -85,B 0,C 180,E1 -16393.616,E2 -16393.616} C_VEL
LIN {X 0,Y 298.547,Z 297.58,A -85,B 0,C 180,E1 -16396.409,E2 -16396.409} C_VEL
LIN {X 0,Y 298.509,Z 297.607,A -85,B 0,C 180,E1 -16399.654,E2 -16399.654} C_VEL
LIN {X 0,Y 298.428,Z 297.607,A -85,B 0,C 180,E1 -16403.6,E2 -16403.6} C_VEL
LIN {X 0,Y 298.486,Z 297.596,A -85,B 0,C 180,E1 -16406.575,E2 -16406.575} C_VEL
LIN {X 0,Y 298.42,Z 297.613,A -85,B 0,C 180,E1 -16409.641,E2 -16409.641} C_VEL
LIN {X 0,Y 298.395,Z 297.625,A -85,B 0,C 180,E1 -16412.8,E2 -16412.8} C_VEL
LIN {X 0,Y 298.443,Z 297.606,A -85,B 0,C 180,E1 -16416.807,E2 -16416.807} C_VEL
LIN {X 0,Y 298.431,Z 297.783,A -85,B 0,C 180,E1 -16419.647,E2 -16419.647} C_VEL
LIN {X 0,Y 299.311,Z 300.319,A -85,B 0,C 180,E1 -16419.945,E2 -16419.945} C_VEL
LIN {X 0,Y 301.356,Z 302.542,A -85,B 0,C 180,E1 -16420.491,E2 -16420.491} C_VEL
LIN {X 0,Y 302.123,Z 303.526,A -85,B 0,C 180,E1 -16420.698,E2 -16420.698} C_VEL
LIN {X 0,Y 304.399,Z 306.826,A -85,B 0,C 180,E1 -16421.313,E2 -16421.313} C_VEL
LIN {X 0,Y 305.707,Z 308.341,A -85,B 0,C 180,E1 -16421.647,E2 -16421.647} C_VEL
LIN {X 0,Y 315.202,Z 321.78,A -85,B 0,C 180,E1 -16424.002,E2 -16424.002} C_VEL
LIN {X 0,Y 324.484,Z 335.79,A -85,B 0,C 180,E1 -16426.112,E2 -16426.112} C_VEL
LIN {X 0,Y 331.827,Z 348.154,A -85,B 0,C 180,E1 -16427.686,E2 -16427.686} C_VEL
LIN {X 0,Y 338.051,Z 360.55,A -85,B 0,C 180,E1 -16428.991,E2 -16428.991} C_VEL
LIN {X 0,Y 332.373,Z 494.939,A -85,B 0,C 180,E1 -16431.889,E2 -16431.889} C_VEL
LIN {X 0,Y 330.979,Z 511.353,A -85,B 0,C 180,E1 -16432.424,E2 -16432.424} C_VEL
LIN {X 0,Y 329.163,Z 527.485,A -85,B 0,C 180,E1 -16433.19,E2 -16433.19} C_VEL
LIN {X 0,Y 326.877,Z 542.793,A -85,B 0,C 180,E1 -16434.135,E2 -16434.135} C_VEL
LIN {X 0,Y 324.212,Z 557.743,A -85,B 0,C 180,E1 -16435.318,E2 -16435.318} C_VEL
LIN {X 0,Y 321.284,Z 571.948,A -85,B 0,C 180,E1 -16436.707,E2 -16436.707} C_VEL
LIN {X 0,Y 318.041,Z 585.807,A -85,B 0,C 180,E1 -16438.344,E2 -16438.344} C_VEL
LIN {X 0,Y 314.714,Z 598.875,A -85,B 0,C 180,E1 -16440.207,E2 -16440.207} C_VEL
LIN {X 0,Y 311.219,Z 611.737,A -85,B 0,C 180,E1 -16442.424,E2 -16442.424} C_VEL
LIN {X 0,Y 308.113,Z 622.582,A -85,B 0,C 180,E1 -16444.679,E2 -16444.679} C_VEL
LIN {X 0,Y 305.383,Z 631.977,A -85,B 0,C 180,E1 -16447.007,E2 -16447.007} C_VEL
LIN {X 0,Y 302.864,Z 640.86,A -85,B 0,C 180,E1 -16449.63,E2 -16449.63} C_VEL
LIN {X 0,Y 300.802,Z 648.387,A -85,B 0,C 180,E1 -16452.318,E2 -16452.318} C_VEL
LIN {X 0,Y 299.196,Z 654.539,A -85,B 0,C 180,E1 -16455.026,E2 -16455.026} C_VEL
LIN {X 0,Y 297.999,Z 659.579,A -85,B 0,C 180,E1 -16457.745,E2 -16457.745} C_VEL
LIN {X 0,Y 297.303,Z 663.472,A -85,B 0,C 180,E1 -16460.475,E2 -16460.475} C_VEL
LIN {X 0,Y 296.864,Z 666.366,A -85,B 0,C 180,E1 -16463.202,E2 -16463.202} C_VEL
LIN {X 0,Y 296.65,Z 668.266,A -85,B 0,C 180,E1 -16465.924,E2 -16465.924} C_VEL
LIN {X 0,Y 296.523,Z 669.229,A -85,B 0,C 180,E1 -16468.642,E2 -16468.642} C_VEL
LIN {X 0,Y 296.523,Z 669.242,A -85,B 0,C 180,E1 -16471.358,E2 -16471.358} C_VEL
LIN {X 0,Y 296.65,Z 668.331,A -85,B 0,C 180,E1 -16474.076,E2 -16474.076} C_VEL
LIN {X 0,Y 296.863,Z 666.458,A -85,B 0,C 180,E1 -16476.798,E2 -16476.798} C_VEL
LIN {X 0,Y 297.284,Z 663.614,A -85,B 0,C 180,E1 -16479.525,E2 -16479.525} C_VEL
LIN {X 0,Y 297.981,Z 659.745,A -85,B 0,C 180,E1 -16482.255,E2 -16482.255} C_VEL
LIN {X 0,Y 299.161,Z 654.764,A -85,B 0,C 180,E1 -16484.976,E2 -16484.976} C_VEL
LIN {X 0,Y 300.772,Z 648.669,A -85,B 0,C 180,E1 -16487.684,E2 -16487.684} C_VEL
LIN {X 0,Y 303.159,Z 640.18,A -85,B 0,C 180,E1 -16490.703,E2 -16490.703} C_VEL
LIN {X 0,Y 305.711,Z 631.014,A -85,B 0,C 180,E1 -16493.363,E2 -16493.363} C_VEL
LIN {X 0,Y 308.463,Z 621.574,A -85,B 0,C 180,E1 -16495.651,E2 -16495.651} C_VEL
LIN {X 0,Y 311.591,Z 610.562,A -85,B 0,C 180,E1 -16497.906,E2 -16497.906} C_VEL
LIN {X 0,Y 314.619,Z 599.485,A -85,B 0,C 180,E1 -16499.803,E2 -16499.803} C_VEL
LIN {X 0,Y 317.914,Z 586.539,A -85,B 0,C 180,E1 -16501.67,E2 -16501.67} C_VEL
LIN {X 0,Y 321.367,Z 572.079,A -85,B 0,C 180,E1 -16503.383,E2 -16503.383} C_VEL
LIN {X 0,Y 323.725,Z 560.449,A -85,B 0,C 180,E1 -16504.553,E2 -16504.553} C_VEL
LIN {X 0,Y 326.377,Z 546.008,A -85,B 0,C 180,E1 -16505.739,E2 -16505.739} C_VEL
LIN {X 0,Y 328.862,Z 530.384,A -85,B 0,C 180,E1 -16506.753,E2 -16506.753} C_VEL
LIN {X 0,Y 330.634,Z 515.409,A -85,B 0,C 180,E1 -16507.526,E2 -16507.526} C_VEL
LIN {X 0,Y 332.256,Z 498.015,A -85,B 0,C 180,E1 -16508.137,E2 -16508.137} C_VEL
LIN {X 0,Y 333.222,Z 477.917,A -85,B 0,C 180,E1 -16508.609,E2 -16508.609} C_VEL
LIN {X 0,Y 332.986,Z 472.119,A -85,B 0,C 180,E1 -16508.799,E2 -16508.799} C_VEL
LIN {X 0,Y 329.184,Z 453.59,A -85,B 0,C 180,E1 -16509.852,E2 -16509.852} C_VEL
LIN {X 0,Y 328.949,Z 447.792,A -85,B 0,C 180,E1 -16510.048,E2 -16510.048} C_VEL
LIN {X 0,Y 332.809,Z 363.383,A -85,B 0,C 180,E1 -16511.847,E2 -16511.847} C_VEL
LIN {X 0,Y 326.619,Z 350.979,A -85,B 0,C 180,E1 -16513.2,E2 -16513.2} C_VEL
LIN {X 0,Y 317.792,Z 336.525,A -85,B 0,C 180,E1 -16515.177,E2 -16515.177} C_VEL
LIN {X 0,Y 309.964,Z 324.871,A -85,B 0,C 180,E1 -16517.05,E2 -16517.05} C_VEL
LIN {X 0,Y 303.959,Z 316.361,A -85,B 0,C 180,E1 -16518.586,E2 -16518.586} C_VEL
LIN {X 0,Y 301.312,Z 312.732,A -85,B 0,C 180,E1 -16519.294,E2 -16519.294} C_VEL
LIN {X 0,Y 298.628,Z 308.924,A -85,B 0,C 180,E1 -16520.04,E2 -16520.04} C_VEL
LIN {X 0,Y 295.785,Z 305.493,A -85,B 0,C 180,E1 -16520.836,E2 -16520.836} C_VEL
LIN {X 0,Y 294.691,Z 303.674,A -85,B 0,C 180,E1 -16521.169,E2 -16521.169} C_VEL
LIN {X 0,Y 292.56,Z 301.623,A -85,B 0,C 180,E1 -16521.774,E2 -16521.774} C_VEL
LIN {X 0,Y 291.495,Z 299.134,A -85,B 0,C 180,E1 -16522.14,E2 -16522.14} C_VEL
LIN {X 0,Y 291.376,Z 298.488,A -85,B 0,C 180,E1 -16522.228,E2 -16522.228} C_VEL
LIN {X 0,Y 291.343,Z 298.492,A -85,B 0,C 180,E1 -16526.301,E2 -16526.301} C_VEL
LIN {X 0,Y 291.382,Z 298.5,A -85,B 0,C 180,E1 -16530.261,E2 -16530.261} C_VEL
LIN {X 0,Y 291.413,Z 298.492,A -85,B 0,C 180,E1 -16534.271,E2 -16534.271} C_VEL
LIN {X 0,Y 291.379,Z 298.475,A -85,B 0,C 180,E1 -16537.299,E2 -16537.299} C_VEL
LIN {X 0,Y 291.456,Z 298.491,A -85,B 0,C 180,E1 -16540.27,E2 -16540.27} C_VEL
LIN {X 0,Y 291.539,Z 298.452,A -85,B 0,C 180,E1 -16544.634,E2 -16544.634} C_VEL
LIN {X 0,Y 291.535,Z 298.462,A -85,B 0,C 180,E1 -16548.88,E2 -16548.88} C_VEL
LIN {X 0,Y 291.707,Z 298.435,A -85,B 0,C 180,E1 -16551.688,E2 -16551.688} C_VEL
LIN {X 0,Y 291.629,Z 298.469,A -85,B 0,C 180,E1 -16554.468,E2 -16554.468} C_VEL
LIN {X 0,Y 291.887,Z 298.415,A -85,B 0,C 180,E1 -16558.62,E2 -16558.62} C_VEL
LIN {X 0,Y 291.888,Z 298.435,A -85,B 0,C 180,E1 -16561.379,E2 -16561.379} C_VEL
LIN {X 0,Y 291.744,Z 298.456,A -85,B 0,C 180,E1 -16566.918,E2 -16566.918} C_VEL
LIN {X 0,Y 291.627,Z 298.443,A -85,B 0,C 180,E1 -16569.712,E2 -16569.712} C_VEL
LIN {X 0,Y 291.52,Z 298.485,A -85,B 0,C 180,E1 -16573.95,E2 -16573.95} C_VEL
LIN {X 0,Y 291.485,Z 298.491,A -85,B 0,C 180,E1 -16576.818,E2 -16576.818} C_VEL
LIN {X 0,Y 291.448,Z 298.496,A -85,B 0,C 180,E1 -16579.875,E2 -16579.875} C_VEL
LIN {X 0,Y 291.398,Z 298.497,A -85,B 0,C 180,E1 -16584.205,E2 -16584.205} C_VEL
LIN {X 0,Y 291.42,Z 298.496,A -85,B 0,C 180,E1 -16587.271,E2 -16587.271} C_VEL
LIN {X 0,Y 291.335,Z 298.507,A -85,B 0,C 180,E1 -16590.437,E2 -16590.437} C_VEL
LIN {X 0,Y 291.343,Z 298.51,A -85,B 0,C 180,E1 -16593.698,E2 -16593.698} C_VEL
LIN {X 0,Y 291.416,Z 298.596,A -85,B 0,C 180,E1 -16596.593,E2 -16596.593} C_VEL
LIN {X 0,Y 293.206,Z 302.96,A -85,B 0,C 180,E1 -16598.073,E2 -16598.073} C_VEL
LIN {X 0,Y 301.766,Z 315.375,A -85,B 0,C 180,E1 -16600.536,E2 -16600.536} C_VEL
LIN {X 0,Y 308.86,Z 326.409,A -85,B 0,C 180,E1 -16602.414,E2 -16602.414} C_VEL
LIN {X 0,Y 316.378,Z 338.803,A -85,B 0,C 180,E1 -16604.27,E2 -16604.27} C_VEL
LIN {X 0,Y 324.14,Z 353.198,A -85,B 0,C 180,E1 -16606.085,E2 -16606.085} C_VEL
LIN {X 0,Y 331.655,Z 368.539,A -85,B 0,C 180,E1 -16607.755,E2 -16607.755} C_VEL
LIN {X 0,Y 332.571,Z 370.65,A -85,B 0,C 180,E1 -16607.957,E2 -16607.957} C_VEL
LIN {X 0,Y 326.302,Z 510.993,A -85,B 0,C 180,E1 -16611.005,E2 -16611.005} C_VEL
LIN {X 0,Y 324.67,Z 527.835,A -85,B 0,C 180,E1 -16611.563,E2 -16611.563} C_VEL
LIN {X 0,Y 322.561,Z 543.626,A -85,B 0,C 180,E1 -16612.307,E2 -16612.307} C_VEL
LIN {X 0,Y 320.125,Z 558.784,A -85,B 0,C 180,E1 -16613.256,E2 -16613.256} C_VEL
LIN {X 0,Y 317.166,Z 573.743,A -85,B 0,C 180,E1 -16614.433,E2 -16614.433} C_VEL
LIN {X 0,Y 313.733,Z 588.999,A -85,B 0,C 180,E1 -16615.942,E2 -16615.942} C_VEL
LIN {X 0,Y 310.227,Z 602.984,A -85,B 0,C 180,E1 -16617.642,E2 -16617.642} C_VEL
LIN {X 0,Y 307.004,Z 614.936,A -85,B 0,C 180,E1 -16619.38,E2 -16619.38} C_VEL
LIN {X 0,Y 303.497,Z 627.293,A -85,B 0,C 180,E1 -16621.522,E2 -16621.522} C_VEL
LIN {X 0,Y 300.107,Z 638.868,A -85,B 0,C 180,E1 -16623.954,E2 -16623.954} C_VEL
LIN {X 0,Y 297.367,Z 648.239,A -85,B 0,C 180,E1 -16626.311,E2 -16626.311} C_VEL
LIN {X 0,Y 294.776,Z 657.379,A -85,B 0,C 180,E1 -16629.046,E2 -16629.046} C_VEL
LIN {X 0,Y 292.781,Z 665.047,A -85,B 0,C 180,E1 -16631.817,E2 -16631.817} C_VEL
LIN {X 0,Y 291.208,Z 671.852,A -85,B 0,C 180,E1 -16634.873,E2 -16634.873} C_VEL
LIN {X 0,Y 290.12,Z 677.534,A -85,B 0,C 180,E1 -16638.118,E2 -16638.118} C_VEL
LIN {X 0,Y 289.672,Z 680.451,A -85,B 0,C 180,E1 -16640.222,E2 -16640.222} C_VEL
LIN {X 0,Y 289.444,Z 683.416,A -85,B 0,C 180,E1 -16643.027,E2 -16643.027} C_VEL
LIN {X 0,Y 289.403,Z 685.372,A -85,B 0,C 180,E1 -16645.822,E2 -16645.822} C_VEL
LIN {X 0,Y 289.409,Z 686.339,A -85,B 0,C 180,E1 -16648.609,E2 -16648.609} C_VEL
LIN {X 0,Y 289.409,Z 686.336,A -85,B 0,C 180,E1 -16651.392,E2 -16651.392} C_VEL
LIN {X 0,Y 289.403,Z 685.358,A -85,B 0,C 180,E1 -16654.178,E2 -16654.178} C_VEL
LIN {X 0,Y 289.445,Z 683.398,A -85,B 0,C 180,E1 -16656.973,E2 -16656.973} C_VEL
LIN {X 0,Y 289.672,Z 680.425,A -85,B 0,C 180,E1 -16659.778,E2 -16659.778} C_VEL
LIN {X 0,Y 290.328,Z 676.422,A -85,B 0,C 180,E1 -16662.584,E2 -16662.584} C_VEL
LIN {X 0,Y 291.309,Z 671.269,A -85,B 0,C 180,E1 -16665.39,E2 -16665.39} C_VEL
LIN {X 0,Y 292.781,Z 664.99,A -85,B 0,C 180,E1 -16668.183,E2 -16668.183} C_VEL
LIN {X 0,Y 294.795,Z 657.313,A -85,B 0,C 180,E1 -16670.953,E2 -16670.953} C_VEL
LIN {X 0,Y 297.361,Z 648.156,A -85,B 0,C 180,E1 -16673.69,E2 -16673.69} C_VEL
LIN {X 0,Y 300.608,Z 637.273,A -85,B 0,C 180,E1 -16676.372,E2 -16676.372} C_VEL
LIN {X 0,Y 303.843,Z 625.838,A -85,B 0,C 180,E1 -16678.725,E2 -16678.725} C_VEL
LIN {X 0,Y 307.214,Z 613.813,A -85,B 0,C 180,E1 -16680.788,E2 -16680.788} C_VEL
LIN {X 0,Y 310.783,Z 600.455,A -85,B 0,C 180,E1 -16682.677,E2 -16682.677} C_VEL
LIN {X 0,Y 314.056,Z 587.356,A -85,B 0,C 180,E1 -16684.211,E2 -16684.211} C_VEL
LIN {X 0,Y 317.155,Z 573.474,A -85,B 0,C 180,E1 -16685.569,E2 -16685.569} C_VEL
LIN {X 0,Y 320.284,Z 557.474,A -85,B 0,C 180,E1 -16686.821,E2 -16686.821} C_VEL
LIN {X 0,Y 322.718,Z 541.931,A -85,B 0,C 180,E1 -16687.77,E2 -16687.77} C_VEL
LIN {X 0,Y 324.868,Z 525.449,A -85,B 0,C 180,E1 -16688.509,E2 -16688.509} C_VEL
LIN {X 0,Y 326.406,Z 508.527,A -85,B 0,C 180,E1 -16689.031,E2 -16689.031} C_VEL
LIN {X 0,Y 332.508,Z 371.066,A -85,B 0,C 180,E1 -16692.009,E2 -16692.009} C_VEL
LIN {X 0,Y 331.168,Z 367.585,A -85,B 0,C 180,E1 -16692.316,E2 -16692.316} C_VEL
LIN {X 0,Y 322.393,Z 349.84,A -85,B 0,C 180,E1 -16694.277,E2 -16694.277} C_VEL
LIN {X 0,Y 315.372,Z 337.196,A -85,B 0,C 180,E1 -16695.927,E2 -16695.927} C_VEL
LIN {X 0,Y 307.089,Z 323.468,A -85,B 0,C 180,E1 -16698,E2 -16698} C_VEL
LIN {X 0,Y 300.391,Z 313.357,A -85,B 0,C 180,E1 -16699.791,E2 -16699.791} C_VEL
LIN {X 0,Y 294.797,Z 305.404,A -85,B 0,C 180,E1 -16701.385,E2 -16701.385} C_VEL
LIN {X 0,Y 293.01,Z 302.499,A -85,B 0,C 180,E1 -16701.95,E2 -16701.95} C_VEL
LIN {X 0,Y 291.392,Z 298.494,A -85,B 0,C 180,E1 -16703.457,E2 -16703.457} C_VEL
LIN {X 0,Y 291.37,Z 298.497,A -85,B 0,C 180,E1 -16707.951,E2 -16707.951} C_VEL
LIN {X 0,Y 291.381,Z 298.502,A -85,B 0,C 180,E1 -16711.159,E2 -16711.159} C_VEL
LIN {X 0,Y 291.415,Z 298.499,A -85,B 0,C 180,E1 -16714.272,E2 -16714.272} C_VEL
LIN {X 0,Y 291.38,Z 298.501,A -85,B 0,C 180,E1 -16717.3,E2 -16717.3} C_VEL
LIN {X 0,Y 291.456,Z 298.459,A -85,B 0,C 180,E1 -16720.27,E2 -16720.27} C_VEL
LIN {X 0,Y 291.539,Z 298.464,A -85,B 0,C 180,E1 -16724.635,E2 -16724.635} C_VEL
LIN {X 0,Y 291.534,Z 298.475,A -85,B 0,C 180,E1 -16728.881,E2 -16728.881} C_VEL
LIN {X 0,Y 291.686,Z 298.443,A -85,B 0,C 180,E1 -16731.688,E2 -16731.688} C_VEL
LIN {X 0,Y 291.626,Z 298.436,A -85,B 0,C 180,E1 -16734.468,E2 -16734.468} C_VEL
LIN {X 0,Y 291.887,Z 298.423,A -85,B 0,C 180,E1 -16738.621,E2 -16738.621} C_VEL
LIN {X 0,Y 291.887,Z 298.4,A -85,B 0,C 180,E1 -16741.38,E2 -16741.38} C_VEL
LIN {X 0,Y 291.734,Z 298.425,A -85,B 0,C 180,E1 -16746.918,E2 -16746.918} C_VEL
LIN {X 0,Y 291.574,Z 298.449,A -85,B 0,C 180,E1 -16749.714,E2 -16749.714} C_VEL
LIN {X 0,Y 291.521,Z 298.456,A -85,B 0,C 180,E1 -16753.951,E2 -16753.951} C_VEL
LIN {X 0,Y 291.486,Z 298.465,A -85,B 0,C 180,E1 -16756.818,E2 -16756.818} C_VEL
LIN {X 0,Y 291.45,Z 298.48,A -85,B 0,C 180,E1 -16759.875,E2 -16759.875} C_VEL
LIN {X 0,Y 291.383,Z 298.497,A -85,B 0,C 180,E1 -16764.207,E2 -16764.207} C_VEL
LIN {X 0,Y 291.42,Z 298.468,A -85,B 0,C 180,E1 -16767.272,E2 -16767.272} C_VEL
LIN {X 0,Y 291.337,Z 298.508,A -85,B 0,C 180,E1 -16770.437,E2 -16770.437} C_VEL
LIN {X 0,Y 291.344,Z 298.504,A -85,B 0,C 180,E1 -16773.699,E2 -16773.699} C_VEL
LIN {X 0,Y 291.37,Z 298.477,A -85,B 0,C 180,E1 -16777.931,E2 -16777.931} C_VEL
LIN {X 0,Y 292.235,Z 301.133,A -85,B 0,C 180,E1 -16778.276,E2 -16778.276} C_VEL
LIN {X 0,Y 294.197,Z 303.334,A -85,B 0,C 180,E1 -16778.846,E2 -16778.846} C_VEL
LIN {X 0,Y 295.064,Z 304.088,A -85,B 0,C 180,E1 -16779.085,E2 -16779.085} C_VEL
LIN {X 0,Y 297.109,Z 307.342,A -85,B 0,C 180,E1 -16779.693,E2 -16779.693} C_VEL
LIN {X 0,Y 298.922,Z 309.434,A -85,B 0,C 180,E1 -16780.19,E2 -16780.19} C_VEL
LIN {X 0,Y 301.532,Z 312.95,A -85,B 0,C 180,E1 -16780.905,E2 -16780.905} C_VEL
LIN {X 0,Y 311.141,Z 326.526,A -85,B 0,C 180,E1 -16783.373,E2 -16783.373} C_VEL
LIN {X 0,Y 320.503,Z 340.829,A -85,B 0,C 180,E1 -16785.574,E2 -16785.574} C_VEL
LIN {X 0,Y 327.441,Z 352.668,A -85,B 0,C 180,E1 -16787.11,E2 -16787.11} C_VEL
LIN {X 0,Y 332.701,Z 363.131,A -85,B 0,C 180,E1 -16788.251,E2 -16788.251} C_VEL
LIN {X 0,Y 326.812,Z 495.527,A -85,B 0,C 180,E1 -16791.132,E2 -16791.132} C_VEL
LIN {X 0,Y 325.395,Z 511.572,A -85,B 0,C 180,E1 -16791.664,E2 -16791.664} C_VEL
LIN {X 0,Y 323.522,Z 527.701,A -85,B 0,C 180,E1 -16792.439,E2 -16792.439} C_VEL
LIN {X 0,Y 321.16,Z 543.007,A -85,B 0,C 180,E1 -16793.394,E2 -16793.394} C_VEL
LIN {X 0,Y 318.399,Z 557.957,A -85,B 0,C 180,E1 -16794.591,E2 -16794.591} C_VEL
LIN {X 0,Y 315.576,Z 571.241,A -85,B 0,C 180,E1 -16795.899,E2 -16795.899} C_VEL
LIN {X 0,Y 312.256,Z 584.854,A -85,B 0,C 180,E1 -16797.496,E2 -16797.496} C_VEL
LIN {X 0,Y 308.842,Z 598.112,A -85,B 0,C 180,E1 -16799.392,E2 -16799.392} C_VEL
LIN {X 0,Y 305.393,Z 610.213,A -85,B 0,C 180,E1 -16801.477,E2 -16801.477} C_VEL
LIN {X 0,Y 302.128,Z 621.318,A -85,B 0,C 180,E1 -16803.77,E2 -16803.77} C_VEL
LIN {X 0,Y 299.212,Z 630.838,A -85,B 0,C 180,E1 -16806.098,E2 -16806.098} C_VEL
LIN {X 0,Y 296.509,Z 640.067,A -85,B 0,C 180,E1 -16808.81,E2 -16808.81} C_VEL
LIN {X 0,Y 293.972,Z 648.598,A -85,B 0,C 180,E1 -16811.893,E2 -16811.893} C_VEL
LIN {X 0,Y 292.298,Z 654.749,A -85,B 0,C 180,E1 -16814.664,E2 -16814.664} C_VEL
LIN {X 0,Y 291.018,Z 659.788,A -85,B 0,C 180,E1 -16817.447,E2 -16817.447} C_VEL
LIN {X 0,Y 290.269,Z 663.681,A -85,B 0,C 180,E1 -16820.242,E2 -16820.242} C_VEL
LIN {X 0,Y 289.785,Z 666.575,A -85,B 0,C 180,E1 -16823.035,E2 -16823.035} C_VEL
LIN {X 0,Y 289.569,Z 668.473,A -85,B 0,C 180,E1 -16825.824,E2 -16825.824} C_VEL
LIN {X 0,Y 289.444,Z 669.435,A -85,B 0,C 180,E1 -16828.609,E2 -16828.609} C_VEL
LIN {X 0,Y 289.444,Z 669.448,A -85,B 0,C 180,E1 -16831.391,E2 -16831.391} C_VEL
LIN {X 0,Y 289.569,Z 668.538,A -85,B 0,C 180,E1 -16834.175,E2 -16834.175} C_VEL
LIN {X 0,Y 289.784,Z 666.665,A -85,B 0,C 180,E1 -16836.965,E2 -16836.965} C_VEL
LIN {X 0,Y 290.252,Z 663.822,A -85,B 0,C 180,E1 -16839.758,E2 -16839.758} C_VEL
LIN {X 0,Y 290.998,Z 659.953,A -85,B 0,C 180,E1 -16842.554,E2 -16842.554} C_VEL
LIN {X 0,Y 292.267,Z 654.971,A -85,B 0,C 180,E1 -16845.338,E2 -16845.338} C_VEL
LIN {X 0,Y 293.941,Z 648.877,A -85,B 0,C 180,E1 -16848.109,E2 -16848.109} C_VEL
LIN {X 0,Y 296.475,Z 640.387,A -85,B 0,C 180,E1 -16851.192,E2 -16851.192} C_VEL
LIN {X 0,Y 299.145,Z 631.222,A -85,B 0,C 180,E1 -16853.907,E2 -16853.907} C_VEL
LIN {X 0,Y 302.042,Z 621.78,A -85,B 0,C 180,E1 -16856.237,E2 -16856.237} C_VEL
LIN {X 0,Y 305.311,Z 610.767,A -85,B 0,C 180,E1 -16858.532,E2 -16858.532} C_VEL
LIN {X 0,Y 308.999,Z 597.727,A -85,B 0,C 180,E1 -16860.78,E2 -16860.78} C_VEL
LIN {X 0,Y 312.495,Z 584.407,A -85,B 0,C 180,E1 -16862.667,E2 -16862.667} C_VEL
LIN {X 0,Y 315.785,Z 570.733,A -85,B 0,C 180,E1 -16864.263,E2 -16864.263} C_VEL
LIN {X 0,Y 318.586,Z 557.287,A -85,B 0,C 180,E1 -16865.579,E2 -16865.579} C_VEL
LIN {X 0,Y 321.406,Z 542.224,A -85,B 0,C 180,E1 -16866.769,E2 -16866.769} C_VEL
LIN {X 0,Y 323.884,Z 525.395,A -85,B 0,C 180,E1 -16867.806,E2 -16867.806} C_VEL
LIN {X 0,Y 325.624,Z 510.141,A -85,B 0,C 180,E1 -16868.501,E2 -16868.501} C_VEL
LIN {X 0,Y 326.976,Z 493.767,A -85,B 0,C 180,E1 -16869.023,E2 -16869.023} C_VEL
LIN {X 0,Y 328.949,Z 447.792,A -85,B 0,C 180,E1 -16870.048,E2 -16870.048} C_VEL
LIN {X 0,Y 328.727,Z 441.991,A -85,B 0,C 180,E1 -16870.244,E2 -16870.244} C_VEL
LIN {X 0,Y 325.131,Z 423.431,A -85,B 0,C 180,E1 -16871.32,E2 -16871.32} C_VEL
LIN {X 0,Y 324.936,Z 417.629,A -85,B 0,C 180,E1 -16871.518,E2 -16871.518} C_VEL
LIN {X 0,Y 327.433,Z 365.655,A -85,B 0,C 180,E1 -16872.634,E2 -16872.634} C_VEL
LIN {X 0,Y 320.938,Z 353.123,A -85,B 0,C 180,E1 -16874.101,E2 -16874.101} C_VEL
LIN {X 0,Y 311.716,Z 338.143,A -85,B 0,C 180,E1 -16876.266,E2 -16876.266} C_VEL
LIN {X 0,Y 303.401,Z 325.989,A -85,B 0,C 180,E1 -16878.368,E2 -16878.368} C_VEL
LIN {X 0,Y 298.091,Z 318.436,A -85,B 0,C 180,E1 -16879.814,E2 -16879.814} C_VEL
LIN {X 0,Y 294.337,Z 313.513,A -85,B 0,C 180,E1 -16880.88,E2 -16880.88} C_VEL
LIN {X 0,Y 291.239,Z 309.351,A -85,B 0,C 180,E1 -16881.803,E2 -16881.803} C_VEL
LIN {X 0,Y 288.842,Z 306.408,A -85,B 0,C 180,E1 -16882.534,E2 -16882.534} C_VEL
LIN {X 0,Y 288.015,Z 304.732,A -85,B 0,C 180,E1 -16882.818,E2 -16882.818} C_VEL
LIN {X 0,Y 285.557,Z 302.548,A -85,B 0,C 180,E1 -16883.569,E2 -16883.569} C_VEL
LIN {X 0,Y 284.478,Z 300.194,A -85,B 0,C 180,E1 -16883.965,E2 -16883.965} C_VEL
LIN {X 0,Y 284.327,Z 299.369,A -85,B 0,C 180,E1 -16884.09,E2 -16884.09} C_VEL
LIN {X 0,Y 284.306,Z 299.362,A -85,B 0,C 180,E1 -16887.189,E2 -16887.189} C_VEL
LIN {X 0,Y 284.354,Z 299.373,A -85,B 0,C 180,E1 -16890.375,E2 -16890.375} C_VEL
LIN {X 0,Y 284.375,Z 299.356,A -85,B 0,C 180,E1 -16893.586,E2 -16893.586} C_VEL
LIN {X 0,Y 284.365,Z 299.354,A -85,B 0,C 180,E1 -16896.707,E2 -16896.707} C_VEL
LIN {X 0,Y 284.402,Z 299.37,A -85,B 0,C 180,E1 -16901.261,E2 -16901.261} C_VEL
LIN {X 0,Y 284.476,Z 299.33,A -85,B 0,C 180,E1 -16904.469,E2 -16904.469} C_VEL
LIN {X 0,Y 284.487,Z 299.344,A -85,B 0,C 180,E1 -16908.601,E2 -16908.601} C_VEL
LIN {X 0,Y 284.657,Z 299.31,A -85,B 0,C 180,E1 -16911.481,E2 -16911.481} C_VEL
LIN {X 0,Y 284.599,Z 299.346,A -85,B 0,C 180,E1 -16914.331,E2 -16914.331} C_VEL
LIN {X 0,Y 284.853,Z 299.29,A -85,B 0,C 180,E1 -16918.586,E2 -16918.586} C_VEL
LIN {X 0,Y 284.854,Z 299.311,A -85,B 0,C 180,E1 -16921.414,E2 -16921.414} C_VEL
LIN {X 0,Y 284.696,Z 299.336,A -85,B 0,C 180,E1 -16927.09,E2 -16927.09} C_VEL
LIN {X 0,Y 284.564,Z 299.32,A -85,B 0,C 180,E1 -16929.955,E2 -16929.955} C_VEL
LIN {X 0,Y 284.48,Z 299.361,A -85,B 0,C 180,E1 -16934.303,E2 -16934.303} C_VEL
LIN {X 0,Y 284.423,Z 299.368,A -85,B 0,C 180,E1 -16937.248,E2 -16937.248} C_VEL
LIN {X 0,Y 284.376,Z 299.378,A -85,B 0,C 180,E1 -16940.242,E2 -16940.242} C_VEL
LIN {X 0,Y 284.367,Z 299.374,A -85,B 0,C 180,E1 -16943.875,E2 -16943.875} C_VEL
LIN {X 0,Y 284.395,Z 299.371,A -85,B 0,C 180,E1 -16947.174,E2 -16947.174} C_VEL
LIN {X 0,Y 284.293,Z 299.39,A -85,B 0,C 180,E1 -16951.274,E2 -16951.274} C_VEL
LIN {X 0,Y 284.352,Z 299.576,A -85,B 0,C 180,E1 -16955.001,E2 -16955.001} C_VEL
LIN {X 0,Y 285.54,Z 302.558,A -85,B 0,C 180,E1 -16956.061,E2 -16956.061} C_VEL
LIN {X 0,Y 290.306,Z 309.125,A -85,B 0,C 180,E1 -16957.586,E2 -16957.586} C_VEL
LIN {X 0,Y 298.149,Z 320.549,A -85,B 0,C 180,E1 -16959.911,E2 -16959.911} C_VEL
LIN {X 0,Y 305.447,Z 332.111,A -85,B 0,C 180,E1 -16961.91,E2 -16961.91} C_VEL
LIN {X 0,Y 312.745,Z 344.3,A -85,B 0,C 180,E1 -16963.766,E2 -16963.766} C_VEL
LIN {X 0,Y 320.861,Z 359.738,A -85,B 0,C 180,E1 -16965.723,E2 -16965.723} C_VEL
LIN {X 0,Y 327.189,Z 372.947,A -85,B 0,C 180,E1 -16967.174,E2 -16967.174} C_VEL
LIN {X 0,Y 320.823,Z 510.815,A -85,B 0,C 180,E1 -16970.209,E2 -16970.209} C_VEL
LIN {X 0,Y 319.221,Z 526.721,A -85,B 0,C 180,E1 -16970.731,E2 -16970.731} C_VEL
LIN {X 0,Y 316.954,Z 543.426,A -85,B 0,C 180,E1 -16971.52,E2 -16971.52} C_VEL
LIN {X 0,Y 314.433,Z 558.582,A -85,B 0,C 180,E1 -16972.478,E2 -16972.478} C_VEL
LIN {X 0,Y 311.381,Z 573.539,A -85,B 0,C 180,E1 -16973.668,E2 -16973.668} C_VEL
LIN {X 0,Y 307.82,Z 588.794,A -85,B 0,C 180,E1 -16975.195,E2 -16975.195} C_VEL
LIN {X 0,Y 304.194,Z 602.778,A -85,B 0,C 180,E1 -16976.919,E2 -16976.919} C_VEL
LIN {X 0,Y 300.811,Z 614.728,A -85,B 0,C 180,E1 -16978.679,E2 -16978.679} C_VEL
LIN {X 0,Y 297.521,Z 625.852,A -85,B 0,C 180,E1 -16980.626,E2 -16980.626} C_VEL
LIN {X 0,Y 294.156,Z 637.166,A -85,B 0,C 180,E1 -16983.003,E2 -16983.003} C_VEL
LIN {X 0,Y 290.772,Z 648.03,A -85,B 0,C 180,E1 -16985.739,E2 -16985.739} C_VEL
LIN {X 0,Y 288.044,Z 657.17,A -85,B 0,C 180,E1 -16988.532,E2 -16988.532} C_VEL
LIN {X 0,Y 285.939,Z 664.838,A -85,B 0,C 180,E1 -16991.366,E2 -16991.366} C_VEL
LIN {X 0,Y 284.2,Z 671.997,A -85,B 0,C 180,E1 -16994.672,E2 -16994.672} C_VEL
LIN {X 0,Y 283.117,Z 677.326,A -85,B 0,C 180,E1 -16997.819,E2 -16997.819} C_VEL
LIN {X 0,Y 282.62,Z 680.243,A -85,B 0,C 180,E1 -16999.976,E2 -16999.976} C_VEL
LIN {X 0,Y 282.345,Z 683.208,A -85,B 0,C 180,E1 -17002.851,E2 -17002.851} C_VEL
LIN {X 0,Y 282.308,Z 685.164,A -85,B 0,C 180,E1 -17005.717,E2 -17005.717} C_VEL
LIN {X 0,Y 282.332,Z 686.132,A -85,B 0,C 180,E1 -17008.574,E2 -17008.574} C_VEL
LIN {X 0,Y 282.332,Z 686.13,A -85,B 0,C 180,E1 -17011.426,E2 -17011.426} C_VEL
LIN {X 0,Y 282.308,Z 685.15,A -85,B 0,C 180,E1 -17014.283,E2 -17014.283} C_VEL
LIN {X 0,Y 282.346,Z 683.189,A -85,B 0,C 180,E1 -17017.149,E2 -17017.149} C_VEL
LIN {X 0,Y 282.62,Z 680.215,A -85,B 0,C 180,E1 -17020.025,E2 -17020.025} C_VEL
LIN {X 0,Y 283.33,Z 676.212,A -85,B 0,C 180,E1 -17022.9,E2 -17022.9} C_VEL
LIN {X 0,Y 284.706,Z 669.615,A -85,B 0,C 180,E1 -17026.492,E2 -17026.492} C_VEL
LIN {X 0,Y 286.429,Z 662.95,A -85,B 0,C 180,E1 -17029.344,E2 -17029.344} C_VEL
LIN {X 0,Y 288.971,Z 654.051,A -85,B 0,C 180,E1 -17032.454,E2 -17032.454} C_VEL
LIN {X 0,Y 291.551,Z 645.456,A -85,B 0,C 180,E1 -17034.951,E2 -17034.951} C_VEL
LIN {X 0,Y 295.119,Z 634.069,A -85,B 0,C 180,E1 -17037.67,E2 -17037.67} C_VEL
LIN {X 0,Y 298.562,Z 622.243,A -85,B 0,C 180,E1 -17040.014,E2 -17040.014} C_VEL
LIN {X 0,Y 302.253,Z 609.339,A -85,B 0,C 180,E1 -17042.133,E2 -17042.133} C_VEL
LIN {X 0,Y 306.006,Z 595.698,A -85,B 0,C 180,E1 -17043.974,E2 -17043.974} C_VEL
LIN {X 0,Y 309.261,Z 582.848,A -85,B 0,C 180,E1 -17045.415,E2 -17045.415} C_VEL
LIN {X 0,Y 312.524,Z 567.948,A -85,B 0,C 180,E1 -17046.779,E2 -17046.779} C_VEL
LIN {X 0,Y 315.371,Z 552.765,A -85,B 0,C 180,E1 -17047.895,E2 -17047.895} C_VEL
LIN {X 0,Y 317.855,Z 536.773,A -85,B 0,C 180,E1 -17048.807,E2 -17048.807} C_VEL
LIN {X 0,Y 319.865,Z 520.517,A -85,B 0,C 180,E1 -17049.48,E2 -17049.48} C_VEL
LIN {X 0,Y 321.12,Z 504.474,A -85,B 0,C 180,E1 -17049.929,E2 -17049.929} C_VEL
LIN {X 0,Y 327.141,Z 372.978,A -85,B 0,C 180,E1 -17052.799,E2 -17052.799} C_VEL
LIN {X 0,Y 319.951,Z 358.084,A -85,B 0,C 180,E1 -17054.448,E2 -17054.448} C_VEL
LIN {X 0,Y 313.666,Z 346.139,A -85,B 0,C 180,E1 -17055.959,E2 -17055.959} C_VEL
LIN {X 0,Y 306.314,Z 333.513,A -85,B 0,C 180,E1 -17057.816,E2 -17057.816} C_VEL
LIN {X 0,Y 300.022,Z 323.412,A -85,B 0,C 180,E1 -17059.511,E2 -17059.511} C_VEL
LIN {X 0,Y 292.294,Z 311.899,A -85,B 0,C 180,E1 -17061.747,E2 -17061.747} C_VEL
LIN {X 0,Y 289.804,Z 308.224,A -85,B 0,C 180,E1 -17062.516,E2 -17062.516} C_VEL
LIN {X 0,Y 286.634,Z 303.983,A -85,B 0,C 180,E1 -17063.517,E2 -17063.517} C_VEL
LIN {X 0,Y 285.213,Z 301.985,A -85,B 0,C 180,E1 -17064.037,E2 -17064.037} C_VEL
LIN {X 0,Y 284.322,Z 299.371,A -85,B 0,C 180,E1 -17065.067,E2 -17065.067} C_VEL
LIN {X 0,Y 284.294,Z 299.384,A -85,B 0,C 180,E1 -17068.726,E2 -17068.726} C_VEL
LIN {X 0,Y 284.396,Z 299.366,A -85,B 0,C 180,E1 -17072.826,E2 -17072.826} C_VEL
LIN {X 0,Y 284.365,Z 299.376,A -85,B 0,C 180,E1 -17076.707,E2 -17076.707} C_VEL
LIN {X 0,Y 284.401,Z 299.345,A -85,B 0,C 180,E1 -17081.262,E2 -17081.262} C_VEL
LIN {X 0,Y 284.476,Z 299.346,A -85,B 0,C 180,E1 -17084.47,E2 -17084.47} C_VEL
LIN {X 0,Y 284.486,Z 299.346,A -85,B 0,C 180,E1 -17088.602,E2 -17088.602} C_VEL
LIN {X 0,Y 284.637,Z 299.324,A -85,B 0,C 180,E1 -17091.481,E2 -17091.481} C_VEL
LIN {X 0,Y 284.596,Z 299.309,A -85,B 0,C 180,E1 -17094.331,E2 -17094.331} C_VEL
LIN {X 0,Y 284.853,Z 299.299,A -85,B 0,C 180,E1 -17098.586,E2 -17098.586} C_VEL
LIN {X 0,Y 284.853,Z 299.275,A -85,B 0,C 180,E1 -17101.414,E2 -17101.414} C_VEL
LIN {X 0,Y 284.685,Z 299.3,A -85,B 0,C 180,E1 -17107.091,E2 -17107.091} C_VEL
LIN {X 0,Y 284.518,Z 299.332,A -85,B 0,C 180,E1 -17109.957,E2 -17109.957} C_VEL
LIN {X 0,Y 284.477,Z 299.328,A -85,B 0,C 180,E1 -17114.303,E2 -17114.303} C_VEL
LIN {X 0,Y 284.424,Z 299.352,A -85,B 0,C 180,E1 -17117.249,E2 -17117.249} C_VEL
LIN {X 0,Y 284.376,Z 299.353,A -85,B 0,C 180,E1 -17120.243,E2 -17120.243} C_VEL
LIN {X 0,Y 284.337,Z 299.381,A -85,B 0,C 180,E1 -17124.847,E2 -17124.847} C_VEL
LIN {X 0,Y 284.329,Z 299.349,A -85,B 0,C 180,E1 -17128.011,E2 -17128.011} C_VEL
LIN {X 0,Y 284.295,Z 299.381,A -85,B 0,C 180,E1 -17131.275,E2 -17131.275} C_VEL
LIN {X 0,Y 284.34,Z 299.375,A -85,B 0,C 180,E1 -17135.348,E2 -17135.348} C_VEL
LIN {X 0,Y 284.338,Z 299.582,A -85,B 0,C 180,E1 -17136.128,E2 -17136.128} C_VEL
LIN {X 0,Y 285.234,Z 302.035,A -85,B 0,C 180,E1 -17136.479,E2 -17136.479} C_VEL
LIN {X 0,Y 287.182,Z 304.181,A -85,B 0,C 180,E1 -17137.093,E2 -17137.093} C_VEL
LIN {X 0,Y 288.185,Z 305.079,A -85,B 0,C 180,E1 -17137.395,E2 -17137.395} C_VEL
LIN {X 0,Y 290.164,Z 308.26,A -85,B 0,C 180,E1 -17138.033,E2 -17138.033} C_VEL
LIN {X 0,Y 292.007,Z 310.226,A -85,B 0,C 180,E1 -17138.573,E2 -17138.573} C_VEL
LIN {X 0,Y 294.693,Z 313.897,A -85,B 0,C 180,E1 -17139.368,E2 -17139.368} C_VEL
LIN {X 0,Y 299.902,Z 321.025,A -85,B 0,C 180,E1 -17140.833,E2 -17140.833} C_VEL
LIN {X 0,Y 308.047,Z 332.711,A -85,B 0,C 180,E1 -17142.964,E2 -17142.964} C_VEL
LIN {X 0,Y 316.646,Z 346.016,A -85,B 0,C 180,E1 -17145.044,E2 -17145.044} C_VEL
LIN {X 0,Y 323.348,Z 357.63,A -85,B 0,C 180,E1 -17146.577,E2 -17146.577} C_VEL
LIN {X 0,Y 327.267,Z 365.438,A -85,B 0,C 180,E1 -17147.457,E2 -17147.457} C_VEL
LIN {X 0,Y 321.304,Z 496.177,A -85,B 0,C 180,E1 -17150.35,E2 -17150.35} C_VEL
LIN {X 0,Y 319.765,Z 512.706,A -85,B 0,C 180,E1 -17150.912,E2 -17150.912} C_VEL
LIN {X 0,Y 317.717,Z 529.214,A -85,B 0,C 180,E1 -17151.73,E2 -17151.73} C_VEL
LIN {X 0,Y 315.108,Z 545.2,A -85,B 0,C 180,E1 -17152.773,E2 -17152.773} C_VEL
LIN {X 0,Y 312.27,Z 559.886,A -85,B 0,C 180,E1 -17153.987,E2 -17153.987} C_VEL
LIN {X 0,Y 308.913,Z 574.863,A -85,B 0,C 180,E1 -17155.534,E2 -17155.534} C_VEL
LIN {X 0,Y 305.41,Z 588.564,A -85,B 0,C 180,E1 -17157.264,E2 -17157.264} C_VEL
LIN {X 0,Y 301.835,Z 601.237,A -85,B 0,C 180,E1 -17159.186,E2 -17159.186} C_VEL
LIN {X 0,Y 298.63,Z 612.16,A -85,B 0,C 180,E1 -17161.155,E2 -17161.155} C_VEL
LIN {X 0,Y 295.261,Z 623.004,A -85,B 0,C 180,E1 -17163.494,E2 -17163.494} C_VEL
LIN {X 0,Y 292.283,Z 632.27,A -85,B 0,C 180,E1 -17165.873,E2 -17165.873} C_VEL
LIN {X 0,Y 289.482,Z 641.281,A -85,B 0,C 180,E1 -17168.644,E2 -17168.644} C_VEL
LIN {X 0,Y 287.185,Z 648.808,A -85,B 0,C 180,E1 -17171.45,E2 -17171.45} C_VEL
LIN {X 0,Y 285.41,Z 654.959,A -85,B 0,C 180,E1 -17174.284,E2 -17174.284} C_VEL
LIN {X 0,Y 284.051,Z 659.998,A -85,B 0,C 180,E1 -17177.134,E2 -17177.134} C_VEL
LIN {X 0,Y 283.25,Z 663.89,A -85,B 0,C 180,E1 -17179.998,E2 -17179.998} C_VEL
LIN {X 0,Y 282.73,Z 666.783,A -85,B 0,C 180,E1 -17182.86,E2 -17182.86} C_VEL
LIN {X 0,Y 282.492,Z 668.681,A -85,B 0,C 180,E1 -17185.72,E2 -17185.72} C_VEL
LIN {X 0,Y 282.368,Z 669.642,A -85,B 0,C 180,E1 -17188.574,E2 -17188.574} C_VEL
LIN {X 0,Y 282.367,Z 669.655,A -85,B 0,C 180,E1 -17191.426,E2 -17191.426} C_VEL
LIN {X 0,Y 282.492,Z 668.745,A -85,B 0,C 180,E1 -17194.28,E2 -17194.28} C_VEL
LIN {X 0,Y 282.729,Z 666.872,A -85,B 0,C 180,E1 -17197.14,E2 -17197.14} C_VEL
LIN {X 0,Y 283.236,Z 664.029,A -85,B 0,C 180,E1 -17200.002,E2 -17200.002} C_VEL
LIN {X 0,Y 284.03,Z 660.161,A -85,B 0,C 180,E1 -17202.867,E2 -17202.867} C_VEL
LIN {X 0,Y 285.379,Z 655.179,A -85,B 0,C 180,E1 -17205.717,E2 -17205.717} C_VEL
LIN {X 0,Y 287.152,Z 649.085,A -85,B 0,C 180,E1 -17208.552,E2 -17208.552} C_VEL
LIN {X 0,Y 289.805,Z 640.595,A -85,B 0,C 180,E1 -17211.704,E2 -17211.704} C_VEL
LIN {X 0,Y 292.597,Z 631.429,A -85,B 0,C 180,E1 -17214.477,E2 -17214.477} C_VEL
LIN {X 0,Y 295.648,Z 621.986,A -85,B 0,C 180,E1 -17216.85,E2 -17216.85} C_VEL
LIN {X 0,Y 299.057,Z 610.973,A -85,B 0,C 180,E1 -17219.185,E2 -17219.185} C_VEL
LIN {X 0,Y 302.306,Z 599.896,A -85,B 0,C 180,E1 -17221.149,E2 -17221.149} C_VEL
LIN {X 0,Y 305.869,Z 586.947,A -85,B 0,C 180,E1 -17223.073,E2 -17223.073} C_VEL
LIN {X 0,Y 309.123,Z 574.311,A -85,B 0,C 180,E1 -17224.637,E2 -17224.637} C_VEL
LIN {X 0,Y 312.12,Z 560.853,A -85,B 0,C 180,E1 -17226.033,E2 -17226.033} C_VEL
LIN {X 0,Y 314.969,Z 546.409,A -85,B 0,C 180,E1 -17227.246,E2 -17227.246} C_VEL
LIN {X 0,Y 317.609,Z 530.781,A -85,B 0,C 180,E1 -17228.285,E2 -17228.285} C_VEL
LIN {X 0,Y 319.421,Z 516.588,A -85,B 0,C 180,E1 -17229.036,E2 -17229.036} C_VEL
LIN {X 0,Y 321.104,Z 500.034,A -85,B 0,C 180,E1 -17229.644,E2 -17229.644} C_VEL
LIN {X 0,Y 322.357,Z 476.507,A -85,B 0,C 180,E1 -17230.219,E2 -17230.219} C_VEL
LIN {X 0,Y 324.936,Z 417.629,A -85,B 0,C 180,E1 -17231.518,E2 -17231.518} C_VEL
LIN {X 0,Y 324.755,Z 411.835,A -85,B 0,C 180,E1 -17231.715,E2 -17231.715} C_VEL
LIN {X 0,Y 321.398,Z 393.277,A -85,B 0,C 180,E1 -17232.807,E2 -17232.807} C_VEL
LIN {X 0,Y 321.231,Z 387.483,A -85,B 0,C 180,E1 -17233.009,E2 -17233.009} C_VEL
LIN {X 0,Y 322.096,Z 368.224,A -85,B 0,C 180,E1 -17233.443,E2 -17233.443} C_VEL
LIN {X 0,Y 316.588,Z 357.548,A -85,B 0,C 180,E1 -17234.734,E2 -17234.734} C_VEL
LIN {X 0,Y 307.814,Z 343.12,A -85,B 0,C 180,E1 -17236.869,E2 -17236.869} C_VEL
LIN {X 0,Y 297.774,Z 328.2,A -85,B 0,C 180,E1 -17239.529,E2 -17239.529} C_VEL
LIN {X 0,Y 291.114,Z 319.115,A -85,B 0,C 180,E1 -17241.453,E2 -17241.453} C_VEL
LIN {X 0,Y 288.003,Z 315.016,A -85,B 0,C 180,E1 -17242.406,E2 -17242.406} C_VEL
LIN {X 0,Y 285.318,Z 311.346,A -85,B 0,C 180,E1 -17243.268,E2 -17243.268} C_VEL
LIN {X 0,Y 282.017,Z 307.47,A -85,B 0,C 180,E1 -17244.349,E2 -17244.349} C_VEL
LIN {X 0,Y 280.891,Z 305.586,A -85,B 0,C 180,E1 -17244.755,E2 -17244.755} C_VEL
LIN {X 0,Y 278.585,Z 303.599,A -85,B 0,C 180,E1 -17245.525,E2 -17245.525} C_VEL
LIN {X 0,Y 277.46,Z 301.355,A -85,B 0,C 180,E1 -17245.97,E2 -17245.97} C_VEL
LIN {X 0,Y 277.246,Z 300.249,A -85,B 0,C 180,E1 -17246.104,E2 -17246.104} C_VEL
LIN {X 0,Y 277.26,Z 300.26,A -85,B 0,C 180,E1 -17249.538,E2 -17249.538} C_VEL
LIN {X 0,Y 277.355,Z 300.224,A -85,B 0,C 180,E1 -17252.864,E2 -17252.864} C_VEL
LIN {X 0,Y 277.327,Z 300.24,A -85,B 0,C 180,E1 -17256.079,E2 -17256.079} C_VEL
LIN {X 0,Y 277.344,Z 300.251,A -85,B 0,C 180,E1 -17260.766,E2 -17260.766} C_VEL
LIN {X 0,Y 277.427,Z 300.215,A -85,B 0,C 180,E1 -17265.325,E2 -17265.325} C_VEL
LIN {X 0,Y 277.505,Z 300.197,A -85,B 0,C 180,E1 -17269.788,E2 -17269.788} C_VEL
LIN {X 0,Y 277.651,Z 300.203,A -85,B 0,C 180,E1 -17272.729,E2 -17272.729} C_VEL
LIN {X 0,Y 277.819,Z 300.164,A -85,B 0,C 180,E1 -17278.55,E2 -17278.55} C_VEL
LIN {X 0,Y 277.82,Z 300.187,A -85,B 0,C 180,E1 -17281.449,E2 -17281.449} C_VEL
LIN {X 0,Y 277.651,Z 300.214,A -85,B 0,C 180,E1 -17287.271,E2 -17287.271} C_VEL
LIN {X 0,Y 277.505,Z 300.197,A -85,B 0,C 180,E1 -17290.211,E2 -17290.211} C_VEL
LIN {X 0,Y 277.433,Z 300.235,A -85,B 0,C 180,E1 -17294.674,E2 -17294.674} C_VEL
LIN {X 0,Y 277.343,Z 300.249,A -85,B 0,C 180,E1 -17299.234,E2 -17299.234} C_VEL
LIN {X 0,Y 277.317,Z 300.251,A -85,B 0,C 180,E1 -17304.17,E2 -17304.17} C_VEL
LIN {X 0,Y 277.324,Z 300.251,A -85,B 0,C 180,E1 -17307.505,E2 -17307.505} C_VEL
LIN {X 0,Y 277.27,Z 300.259,A -85,B 0,C 180,E1 -17310.481,E2 -17310.481} C_VEL
LIN {X 0,Y 277.25,Z 300.292,A -85,B 0,C 180,E1 -17313.17,E2 -17313.17} C_VEL
LIN {X 0,Y 277.818,Z 302.276,A -85,B 0,C 180,E1 -17313.816,E2 -17313.816} C_VEL
LIN {X 0,Y 279.442,Z 304.564,A -85,B 0,C 180,E1 -17314.408,E2 -17314.408} C_VEL
LIN {X 0,Y 280.793,Z 306.079,A -85,B 0,C 180,E1 -17314.873,E2 -17314.873} C_VEL
LIN {X 0,Y 284.042,Z 310.474,A -85,B 0,C 180,E1 -17315.981,E2 -17315.981} C_VEL
LIN {X 0,Y 287.176,Z 314.821,A -85,B 0,C 180,E1 -17317.004,E2 -17317.004} C_VEL
LIN {X 0,Y 292.864,Z 323.216,A -85,B 0,C 180,E1 -17318.769,E2 -17318.769} C_VEL
LIN {X 0,Y 299.255,Z 333.078,A -85,B 0,C 180,E1 -17320.615,E2 -17320.615} C_VEL
LIN {X 0,Y 306.686,Z 345.595,A -85,B 0,C 180,E1 -17322.622,E2 -17322.622} C_VEL
LIN {X 0,Y 313.114,Z 357.341,A -85,B 0,C 180,E1 -17324.256,E2 -17324.256} C_VEL
LIN {X 0,Y 321.901,Z 375.369,A -85,B 0,C 180,E1 -17326.374,E2 -17326.374} C_VEL
LIN {X 0,Y 315.397,Z 510.625,A -85,B 0,C 180,E1 -17329.383,E2 -17329.383} C_VEL
LIN {X 0,Y 313.756,Z 526.525,A -85,B 0,C 180,E1 -17329.911,E2 -17329.911} C_VEL
LIN {X 0,Y 311.413,Z 543.226,A -85,B 0,C 180,E1 -17330.705,E2 -17330.705} C_VEL
LIN {X 0,Y 308.81,Z 558.379,A -85,B 0,C 180,E1 -17331.672,E2 -17331.672} C_VEL
LIN {X 0,Y 305.671,Z 573.337,A -85,B 0,C 180,E1 -17332.877,E2 -17332.877} C_VEL
LIN {X 0,Y 301.996,Z 588.591,A -85,B 0,C 180,E1 -17334.424,E2 -17334.424} C_VEL
LIN {X 0,Y 298.193,Z 602.572,A -85,B 0,C 180,E1 -17336.165,E2 -17336.165} C_VEL
LIN {X 0,Y 294.674,Z 614.521,A -85,B 0,C 180,E1 -17337.95,E2 -17337.95} C_VEL
LIN {X 0,Y 291.191,Z 625.886,A -85,B 0,C 180,E1 -17339.977,E2 -17339.977} C_VEL
LIN {X 0,Y 287.772,Z 636.959,A -85,B 0,C 180,E1 -17342.354,E2 -17342.354} C_VEL
LIN {X 0,Y 284.211,Z 647.821,A -85,B 0,C 180,E1 -17345.142,E2 -17345.142} C_VEL
LIN {X 0,Y 281.346,Z 656.961,A -85,B 0,C 180,E1 -17347.995,E2 -17347.995} C_VEL
LIN {X 0,Y 279.105,Z 664.629,A -85,B 0,C 180,E1 -17350.892,E2 -17350.892} C_VEL
LIN {X 0,Y 277.177,Z 672.171,A -85,B 0,C 180,E1 -17354.474,E2 -17354.474} C_VEL
LIN {X 0,Y 275.87,Z 678.197,A -85,B 0,C 180,E1 -17358.241,E2 -17358.241} C_VEL
LIN {X 0,Y 275.364,Z 681.633,A -85,B 0,C 180,E1 -17361.191,E2 -17361.191} C_VEL
LIN {X 0,Y 275.228,Z 684.136,A -85,B 0,C 180,E1 -17364.138,E2 -17364.138} C_VEL
LIN {X 0,Y 275.24,Z 685.55,A -85,B 0,C 180,E1 -17367.073,E2 -17367.073} C_VEL
LIN {X 0,Y 275.275,Z 686.081,A -85,B 0,C 180,E1 -17370,E2 -17370} C_VEL
LIN {X 0,Y 275.24,Z 685.541,A -85,B 0,C 180,E1 -17372.927,E2 -17372.927} C_VEL
LIN {X 0,Y 275.228,Z 684.119,A -85,B 0,C 180,E1 -17375.862,E2 -17375.862} C_VEL
LIN {X 0,Y 275.364,Z 681.608,A -85,B 0,C 180,E1 -17378.809,E2 -17378.809} C_VEL
LIN {X 0,Y 275.869,Z 678.164,A -85,B 0,C 180,E1 -17381.76,E2 -17381.76} C_VEL
LIN {X 0,Y 277.173,Z 672.131,A -85,B 0,C 180,E1 -17385.523,E2 -17385.523} C_VEL
LIN {X 0,Y 279.107,Z 664.566,A -85,B 0,C 180,E1 -17389.108,E2 -17389.108} C_VEL
LIN {X 0,Y 281.377,Z 656.889,A -85,B 0,C 180,E1 -17392.003,E2 -17392.003} C_VEL
LIN {X 0,Y 284.208,Z 647.731,A -85,B 0,C 180,E1 -17394.859,E2 -17394.859} C_VEL
LIN {X 0,Y 287.819,Z 636.85,A -85,B 0,C 180,E1 -17397.642,E2 -17397.642} C_VEL
LIN {X 0,Y 291.244,Z 625.617,A -85,B 0,C 180,E1 -17400.047,E2 -17400.047} C_VEL
LIN {X 0,Y 294.966,Z 613.388,A -85,B 0,C 180,E1 -17402.216,E2 -17402.216} C_VEL
LIN {X 0,Y 298.51,Z 601.209,A -85,B 0,C 180,E1 -17403.997,E2 -17403.997} C_VEL
LIN {X 0,Y 301.981,Z 588.363,A -85,B 0,C 180,E1 -17405.579,E2 -17405.579} C_VEL
LIN {X 0,Y 305.656,Z 573.046,A -85,B 0,C 180,E1 -17407.126,E2 -17407.126} C_VEL
LIN {X 0,Y 308.996,Z 557.046,A -85,B 0,C 180,E1 -17408.404,E2 -17408.404} C_VEL
LIN {X 0,Y 311.612,Z 541.501,A -85,B 0,C 180,E1 -17409.369,E2 -17409.369} C_VEL
LIN {X 0,Y 313.882,Z 525.013,A -85,B 0,C 180,E1 -17410.123,E2 -17410.123} C_VEL
LIN {X 0,Y 315.459,Z 508.329,A -85,B 0,C 180,E1 -17410.653,E2 -17410.653} C_VEL
LIN {X 0,Y 321.815,Z 375.383,A -85,B 0,C 180,E1 -17413.604,E2 -17413.604} C_VEL
LIN {X 0,Y 313.78,Z 358.715,A -85,B 0,C 180,E1 -17415.535,E2 -17415.535} C_VEL
LIN {X 0,Y 307.008,Z 346.215,A -85,B 0,C 180,E1 -17417.246,E2 -17417.246} C_VEL
LIN {X 0,Y 299.261,Z 333.103,A -85,B 0,C 180,E1 -17419.331,E2 -17419.331} C_VEL
LIN {X 0,Y 292.959,Z 323.435,A -85,B 0,C 180,E1 -17421.142,E2 -17421.142} C_VEL
LIN {X 0,Y 288.305,Z 316.567,A -85,B 0,C 180,E1 -17422.569,E2 -17422.569} C_VEL
LIN {X 0,Y 285.744,Z 312.809,A -85,B 0,C 180,E1 -17423.393,E2 -17423.393} C_VEL
LIN {X 0,Y 281.744,Z 307.363,A -85,B 0,C 180,E1 -17424.727,E2 -17424.727} C_VEL
LIN {X 0,Y 279.631,Z 304.723,A -85,B 0,C 180,E1 -17425.455,E2 -17425.455} C_VEL
LIN {X 0,Y 277.877,Z 302.414,A -85,B 0,C 180,E1 -17426.083,E2 -17426.083} C_VEL
LIN {X 0,Y 277.49,Z 301.444,A -85,B 0,C 180,E1 -17426.338,E2 -17426.338} C_VEL
LIN {X 0,Y 277.252,Z 300.255,A -85,B 0,C 180,E1 -17426.773,E2 -17426.773} C_VEL
LIN {X 0,Y 277.288,Z 300.257,A -85,B 0,C 180,E1 -17431.213,E2 -17431.213} C_VEL
LIN {X 0,Y 277.312,Z 300.254,A -85,B 0,C 180,E1 -17434.48,E2 -17434.48} C_VEL
LIN {X 0,Y 277.284,Z 300.252,A -85,B 0,C 180,E1 -17437.655,E2 -17437.655} C_VEL
LIN {X 0,Y 277.343,Z 300.218,A -85,B 0,C 180,E1 -17440.766,E2 -17440.766} C_VEL
LIN {X 0,Y 277.426,Z 300.208,A -85,B 0,C 180,E1 -17445.326,E2 -17445.326} C_VEL
LIN {X 0,Y 277.46,Z 300.237,A -85,B 0,C 180,E1 -17449.787,E2 -17449.787} C_VEL
LIN {X 0,Y 277.639,Z 300.175,A -85,B 0,C 180,E1 -17452.729,E2 -17452.729} C_VEL
LIN {X 0,Y 277.819,Z 300.176,A -85,B 0,C 180,E1 -17458.551,E2 -17458.551} C_VEL
LIN {X 0,Y 277.819,Z 300.15,A -85,B 0,C 180,E1 -17461.45,E2 -17461.45} C_VEL
LIN {X 0,Y 277.64,Z 300.174,A -85,B 0,C 180,E1 -17467.271,E2 -17467.271} C_VEL
LIN {X 0,Y 277.46,Z 300.215,A -85,B 0,C 180,E1 -17470.213,E2 -17470.213} C_VEL
LIN {X 0,Y 277.427,Z 300.202,A -85,B 0,C 180,E1 -17474.675,E2 -17474.675} C_VEL
LIN {X 0,Y 277.344,Z 300.248,A -85,B 0,C 180,E1 -17479.234,E2 -17479.234} C_VEL
LIN {X 0,Y 277.291,Z 300.248,A -85,B 0,C 180,E1 -17484.158,E2 -17484.158} C_VEL
LIN {X 0,Y 277.324,Z 300.222,A -85,B 0,C 180,E1 -17487.505,E2 -17487.505} C_VEL
LIN {X 0,Y 277.271,Z 300.26,A -85,B 0,C 180,E1 -17490.482,E2 -17490.482} C_VEL
LIN {X 0,Y 277.249,Z 300.256,A -85,B 0,C 180,E1 -17494.06,E2 -17494.06} C_VEL
LIN {X 0,Y 278.155,Z 302.939,A -85,B 0,C 180,E1 -17494.481,E2 -17494.481} C_VEL
LIN {X 0,Y 280.297,Z 305.214,A -85,B 0,C 180,E1 -17495.218,E2 -17495.218} C_VEL
LIN {X 0,Y 281.323,Z 306.09,A -85,B 0,C 180,E1 -17495.554,E2 -17495.554} C_VEL
LIN {X 0,Y 283.342,Z 309.271,A -85,B 0,C 180,E1 -17496.26,E2 -17496.26} C_VEL
LIN {X 0,Y 285.305,Z 311.338,A -85,B 0,C 180,E1 -17496.884,E2 -17496.884} C_VEL
LIN {X 0,Y 287.855,Z 314.844,A -85,B 0,C 180,E1 -17497.702,E2 -17497.702} C_VEL
LIN {X 0,Y 289.345,Z 316.74,A -85,B 0,C 180,E1 -17498.16,E2 -17498.16} C_VEL
LIN {X 0,Y 293.081,Z 321.839,A -85,B 0,C 180,E1 -17499.283,E2 -17499.283} C_VEL
LIN {X 0,Y 298.2,Z 328.832,A -85,B 0,C 180,E1 -17500.734,E2 -17500.734} C_VEL
LIN {X 0,Y 308.277,Z 343.885,A -85,B 0,C 180,E1 -17503.385,E2 -17503.385} C_VEL
LIN {X 0,Y 317.401,Z 359.07,A -85,B 0,C 180,E1 -17505.589,E2 -17505.589} C_VEL
LIN {X 0,Y 321.983,Z 368.038,A -85,B 0,C 180,E1 -17506.659,E2 -17506.659} C_VEL
LIN {X 0,Y 315.943,Z 495.497,A -85,B 0,C 180,E1 -17509.508,E2 -17509.508} C_VEL
LIN {X 0,Y 314.416,Z 512.01,A -85,B 0,C 180,E1 -17510.064,E2 -17510.064} C_VEL
LIN {X 0,Y 312.386,Z 528.133,A -85,B 0,C 180,E1 -17510.851,E2 -17510.851} C_VEL
LIN {X 0,Y 309.89,Z 543.434,A -85,B 0,C 180,E1 -17511.83,E2 -17511.83} C_VEL
LIN {X 0,Y 307.263,Z 556.625,A -85,B 0,C 180,E1 -17512.896,E2 -17512.896} C_VEL
LIN {X 0,Y 304.225,Z 570.255,A -85,B 0,C 180,E1 -17514.236,E2 -17514.236} C_VEL
LIN {X 0,Y 300.681,Z 584.11,A -85,B 0,C 180,E1 -17515.878,E2 -17515.878} C_VEL
LIN {X 0,Y 296.942,Z 597.491,A -85,B 0,C 180,E1 -17517.824,E2 -17517.824} C_VEL
LIN {X 0,Y 293.491,Z 608.866,A -85,B 0,C 180,E1 -17519.81,E2 -17519.81} C_VEL
LIN {X 0,Y 289.878,Z 620.266,A -85,B 0,C 180,E1 -17522.179,E2 -17522.179} C_VEL
LIN {X 0,Y 286.573,Z 630.03,A -85,B 0,C 180,E1 -17524.585,E2 -17524.585} C_VEL
LIN {X 0,Y 283.556,Z 639.392,A -85,B 0,C 180,E1 -17527.408,E2 -17527.408} C_VEL
LIN {X 0,Y 280.945,Z 647.231,A -85,B 0,C 180,E1 -17530.263,E2 -17530.263} C_VEL
LIN {X 0,Y 278.944,Z 653.876,A -85,B 0,C 180,E1 -17533.218,E2 -17533.218} C_VEL
LIN {X 0,Y 277.466,Z 659.044,A -85,B 0,C 180,E1 -17536.076,E2 -17536.076} C_VEL
LIN {X 0,Y 276.607,Z 662.307,A -85,B 0,C 180,E1 -17538.272,E2 -17538.272} C_VEL
LIN {X 0,Y 275.901,Z 665.658,A -85,B 0,C 180,E1 -17541.209,E2 -17541.209} C_VEL
LIN {X 0,Y 275.485,Z 668.153,A -85,B 0,C 180,E1 -17544.236,E2 -17544.236} C_VEL
LIN {X 0,Y 275.354,Z 669.472,A -85,B 0,C 180,E1 -17547.074,E2 -17547.074} C_VEL
LIN {X 0,Y 275.283,Z 670.004,A -85,B 0,C 180,E1 -17550,E2 -17550} C_VEL
LIN {X 0,Y 275.353,Z 669.51,A -85,B 0,C 180,E1 -17552.926,E2 -17552.926} C_VEL
LIN {X 0,Y 275.493,Z 668.168,A -85,B 0,C 180,E1 -17555.857,E2 -17555.857} C_VEL
LIN {X 0,Y 275.894,Z 665.771,A -85,B 0,C 180,E1 -17558.791,E2 -17558.791} C_VEL
LIN {X 0,Y 276.588,Z 662.466,A -85,B 0,C 180,E1 -17561.728,E2 -17561.728} C_VEL
LIN {X 0,Y 278.095,Z 656.78,A -85,B 0,C 180,E1 -17565.388,E2 -17565.388} C_VEL
LIN {X 0,Y 280.362,Z 649.293,A -85,B 0,C 180,E1 -17569.019,E2 -17569.019} C_VEL
LIN {X 0,Y 283.154,Z 640.802,A -85,B 0,C 180,E1 -17572.241,E2 -17572.241} C_VEL
LIN {X 0,Y 286.079,Z 631.637,A -85,B 0,C 180,E1 -17575.073,E2 -17575.073} C_VEL
LIN {X 0,Y 289.277,Z 622.193,A -85,B 0,C 180,E1 -17577.49,E2 -17577.49} C_VEL
LIN {X 0,Y 292.849,Z 611.178,A -85,B 0,C 180,E1 -17579.866,E2 -17579.866} C_VEL
LIN {X 0,Y 296.221,Z 600.101,A -85,B 0,C 180,E1 -17581.863,E2 -17581.863} C_VEL
LIN {X 0,Y 299.915,Z 587.151,A -85,B 0,C 180,E1 -17583.817,E2 -17583.817} C_VEL
LIN {X 0,Y 303.29,Z 574.515,A -85,B 0,C 180,E1 -17585.402,E2 -17585.402} C_VEL
LIN {X 0,Y 306.397,Z 561.055,A -85,B 0,C 180,E1 -17586.815,E2 -17586.815} C_VEL
LIN {X 0,Y 309.348,Z 546.609,A -85,B 0,C 180,E1 -17588.042,E2 -17588.042} C_VEL
LIN {X 0,Y 312.068,Z 530.979,A -85,B 0,C 180,E1 -17589.093,E2 -17589.093} C_VEL
LIN {X 0,Y 313.948,Z 516.785,A -85,B 0,C 180,E1 -17589.851,E2 -17589.851} C_VEL
LIN {X 0,Y 315.712,Z 499.731,A -85,B 0,C 180,E1 -17590.482,E2 -17590.482} C_VEL
LIN {X 0,Y 317.077,Z 473.957,A -85,B 0,C 180,E1 -17591.111,E2 -17591.111} C_VEL
LIN {X 0,Y 321.231,Z 387.483,A -85,B 0,C 180,E1 -17593.009,E2 -17593.009} C_VEL
LIN {X 0,Y 320.925,Z 382.31,A -85,B 0,C 180,E1 -17593.216,E2 -17593.216} C_VEL
LIN {X 0,Y 319.694,Z 377.494,A -85,B 0,C 180,E1 -17593.571,E2 -17593.571} C_VEL
LIN {X 0,Y 317.885,Z 372.967,A -85,B 0,C 180,E1 -17594.024,E2 -17594.024} C_VEL
LIN {X 0,Y 315.834,Z 368.672,A -85,B 0,C 180,E1 -17594.521,E2 -17594.521} C_VEL
LIN {X 0,Y 310.577,Z 358.97,A -85,B 0,C 180,E1 -17595.805,E2 -17595.805} C_VEL
LIN {X 0,Y 301.888,Z 344.904,A -85,B 0,C 180,E1 -17598.029,E2 -17598.029} C_VEL
LIN {X 0,Y 291.856,Z 330.011,A -85,B 0,C 180,E1 -17600.849,E2 -17600.849} C_VEL
LIN {X 0,Y 284.692,Z 320.471,A -85,B 0,C 180,E1 -17603.06,E2 -17603.06} C_VEL
LIN {X 0,Y 281.428,Z 316.149,A -85,B 0,C 180,E1 -17604.144,E2 -17604.144} C_VEL
LIN {X 0,Y 278.783,Z 312.745,A -85,B 0,C 180,E1 -17605.059,E2 -17605.059} C_VEL
LIN {X 0,Y 278.016,Z 311.686,A -85,B 0,C 180,E1 -17605.335,E2 -17605.335} C_VEL
LIN {X 0,Y 275.393,Z 308.89,A -85,B 0,C 180,E1 -17606.266,E2 -17606.266} C_VEL
LIN {X 0,Y 274.158,Z 306.612,A -85,B 0,C 180,E1 -17606.765,E2 -17606.765} C_VEL
LIN {X 0,Y 271.731,Z 304.708,A -85,B 0,C 180,E1 -17607.652,E2 -17607.652} C_VEL
LIN {X 0,Y 270.468,Z 302.343,A -85,B 0,C 180,E1 -17608.197,E2 -17608.197} C_VEL
LIN {X 0,Y 270.185,Z 301.124,A -85,B 0,C 180,E1 -17608.379,E2 -17608.379} C_VEL
LIN {X 0,Y 270.262,Z 301.106,A -85,B 0,C 180,E1 -17612.146,E2 -17612.146} C_VEL
LIN {X 0,Y 270.276,Z 301.129,A -85,B 0,C 180,E1 -17615.519,E2 -17615.519} C_VEL
LIN {X 0,Y 270.3,Z 301.123,A -85,B 0,C 180,E1 -17620.244,E2 -17620.244} C_VEL
LIN {X 0,Y 270.395,Z 301.086,A -85,B 0,C 180,E1 -17624.935,E2 -17624.935} C_VEL
LIN {X 0,Y 270.44,Z 301.078,A -85,B 0,C 180,E1 -17629.519,E2 -17629.519} C_VEL
LIN {X 0,Y 270.609,Z 301.074,A -85,B 0,C 180,E1 -17632.539,E2 -17632.539} C_VEL
LIN {X 0,Y 270.785,Z 301.039,A -85,B 0,C 180,E1 -17638.513,E2 -17638.513} C_VEL
LIN {X 0,Y 270.785,Z 301.061,A -85,B 0,C 180,E1 -17641.487,E2 -17641.487} C_VEL
LIN {X 0,Y 270.609,Z 301.09,A -85,B 0,C 180,E1 -17647.461,E2 -17647.461} C_VEL
LIN {X 0,Y 270.44,Z 301.076,A -85,B 0,C 180,E1 -17650.481,E2 -17650.481} C_VEL
LIN {X 0,Y 270.401,Z 301.109,A -85,B 0,C 180,E1 -17655.064,E2 -17655.064} C_VEL
LIN {X 0,Y 270.299,Z 301.131,A -85,B 0,C 180,E1 -17659.755,E2 -17659.755} C_VEL
LIN {X 0,Y 270.272,Z 301.129,A -85,B 0,C 180,E1 -17664.585,E2 -17664.585} C_VEL
LIN {X 0,Y 270.27,Z 301.132,A -85,B 0,C 180,E1 -17667.908,E2 -17667.908} C_VEL
LIN {X 0,Y 270.215,Z 301.311,A -85,B 0,C 180,E1 -17671.267,E2 -17671.267} C_VEL
LIN {X 0,Y 271.189,Z 303.951,A -85,B 0,C 180,E1 -17671.763,E2 -17671.763} C_VEL
LIN {X 0,Y 273.09,Z 305.998,A -85,B 0,C 180,E1 -17672.494,E2 -17672.494} C_VEL
LIN {X 0,Y 274.44,Z 307.141,A -85,B 0,C 180,E1 -17672.985,E2 -17672.985} C_VEL
LIN {X 0,Y 276.448,Z 310.291,A -85,B 0,C 180,E1 -17673.76,E2 -17673.76} C_VEL
LIN {X 0,Y 278.165,Z 312.244,A -85,B 0,C 180,E1 -17674.369,E2 -17674.369} C_VEL
LIN {X 0,Y 281.733,Z 317.228,A -85,B 0,C 180,E1 -17675.623,E2 -17675.623} C_VEL
LIN {X 0,Y 284.447,Z 321.089,A -85,B 0,C 180,E1 -17676.534,E2 -17676.534} C_VEL
LIN {X 0,Y 289.267,Z 328.242,A -85,B 0,C 180,E1 -17678.077,E2 -17678.077} C_VEL
LIN {X 0,Y 295.634,Z 338.239,A -85,B 0,C 180,E1 -17679.986,E2 -17679.986} C_VEL
LIN {X 0,Y 303.56,Z 351.816,A -85,B 0,C 180,E1 -17682.196,E2 -17682.196} C_VEL
LIN {X 0,Y 310.131,Z 364.228,A -85,B 0,C 180,E1 -17683.916,E2 -17683.916} C_VEL
LIN {X 0,Y 316.644,Z 377.875,A -85,B 0,C 180,E1 -17685.544,E2 -17685.544} C_VEL
LIN {X 0,Y 310.036,Z 510.419,A -85,B 0,C 180,E1 -17688.527,E2 -17688.527} C_VEL
LIN {X 0,Y 308.242,Z 527.245,A -85,B 0,C 180,E1 -17689.096,E2 -17689.096} C_VEL
LIN {X 0,Y 305.945,Z 543.026,A -85,B 0,C 180,E1 -17689.862,E2 -17689.862} C_VEL
LIN {X 0,Y 303.257,Z 558.177,A -85,B 0,C 180,E1 -17690.838,E2 -17690.838} C_VEL
LIN {X 0,Y 300.012,Z 573.134,A -85,B 0,C 180,E1 -17692.054,E2 -17692.054} C_VEL
LIN {X 0,Y 296.217,Z 588.386,A -85,B 0,C 180,E1 -17693.62,E2 -17693.62} C_VEL
LIN {X 0,Y 292.295,Z 602.367,A -85,B 0,C 180,E1 -17695.386,E2 -17695.386} C_VEL
LIN {X 0,Y 288.601,Z 614.314,A -85,B 0,C 180,E1 -17697.192,E2 -17697.192} C_VEL
LIN {X 0,Y 285.015,Z 625.546,A -85,B 0,C 180,E1 -17699.226,E2 -17699.226} C_VEL
LIN {X 0,Y 281.416,Z 636.751,A -85,B 0,C 180,E1 -17701.674,E2 -17701.674} C_VEL
LIN {X 0,Y 277.679,Z 647.612,A -85,B 0,C 180,E1 -17704.516,E2 -17704.516} C_VEL
LIN {X 0,Y 274.666,Z 656.751,A -85,B 0,C 180,E1 -17707.43,E2 -17707.43} C_VEL
LIN {X 0,Y 272.298,Z 664.419,A -85,B 0,C 180,E1 -17710.395,E2 -17710.395} C_VEL
LIN {X 0,Y 270.543,Z 670.684,A -85,B 0,C 180,E1 -17713.396,E2 -17713.396} C_VEL
LIN {X 0,Y 269.315,Z 675.825,A -85,B 0,C 180,E1 -17716.417,E2 -17716.417} C_VEL
LIN {X 0,Y 268.502,Z 679.825,A -85,B 0,C 180,E1 -17719.443,E2 -17719.443} C_VEL
LIN {X 0,Y 268.174,Z 682.792,A -85,B 0,C 180,E1 -17722.471,E2 -17722.471} C_VEL
LIN {X 0,Y 268.134,Z 684.75,A -85,B 0,C 180,E1 -17725.49,E2 -17725.49} C_VEL
LIN {X 0,Y 268.182,Z 685.719,A -85,B 0,C 180,E1 -17728.498,E2 -17728.498} C_VEL
LIN {X 0,Y 268.182,Z 685.716,A -85,B 0,C 180,E1 -17731.502,E2 -17731.502} C_VEL
LIN {X 0,Y 268.134,Z 684.735,A -85,B 0,C 180,E1 -17734.51,E2 -17734.51} C_VEL
LIN {X 0,Y 268.174,Z 682.771,A -85,B 0,C 180,E1 -17737.529,E2 -17737.529} C_VEL
LIN {X 0,Y 268.502,Z 679.795,A -85,B 0,C 180,E1 -17740.558,E2 -17740.558} C_VEL
LIN {X 0,Y 269.309,Z 675.79,A -85,B 0,C 180,E1 -17743.584,E2 -17743.584} C_VEL
LIN {X 0,Y 270.539,Z 670.635,A -85,B 0,C 180,E1 -17746.604,E2 -17746.604} C_VEL
LIN {X 0,Y 272.3,Z 664.354,A -85,B 0,C 180,E1 -17749.604,E2 -17749.604} C_VEL
LIN {X 0,Y 274.712,Z 656.677,A -85,B 0,C 180,E1 -17752.566,E2 -17752.566} C_VEL
LIN {X 0,Y 277.684,Z 647.519,A -85,B 0,C 180,E1 -17755.484,E2 -17755.484} C_VEL
LIN {X 0,Y 281.463,Z 636.638,A -85,B 0,C 180,E1 -17758.322,E2 -17758.322} C_VEL
LIN {X 0,Y 284.479,Z 627.147,A -85,B 0,C 180,E1 -17760.427,E2 -17760.427} C_VEL
LIN {X 0,Y 287.985,Z 616.118,A -85,B 0,C 180,E1 -17762.472,E2 -17762.472} C_VEL
LIN {X 0,Y 291.883,Z 603.352,A -85,B 0,C 180,E1 -17764.46,E2 -17764.46} C_VEL
LIN {X 0,Y 295.914,Z 589.202,A -85,B 0,C 180,E1 -17766.268,E2 -17766.268} C_VEL
LIN {X 0,Y 299.603,Z 574.521,A -85,B 0,C 180,E1 -17767.794,E2 -17767.794} C_VEL
LIN {X 0,Y 302.831,Z 559.827,A -85,B 0,C 180,E1 -17769.013,E2 -17769.013} C_VEL
LIN {X 0,Y 305.693,Z 543.889,A -85,B 0,C 180,E1 -17770.07,E2 -17770.07} C_VEL
LIN {X 0,Y 308.149,Z 527.546,A -85,B 0,C 180,E1 -17770.865,E2 -17770.865} C_VEL
LIN {X 0,Y 309.944,Z 510.811,A -85,B 0,C 180,E1 -17771.437,E2 -17771.437} C_VEL
LIN {X 0,Y 316.544,Z 377.861,A -85,B 0,C 180,E1 -17774.435,E2 -17774.435} C_VEL
LIN {X 0,Y 308.283,Z 360.661,A -85,B 0,C 180,E1 -17776.513,E2 -17776.513} C_VEL
LIN {X 0,Y 300.016,Z 345.598,A -85,B 0,C 180,E1 -17778.721,E2 -17778.721} C_VEL
LIN {X 0,Y 292.913,Z 333.905,A -85,B 0,C 180,E1 -17780.756,E2 -17780.756} C_VEL
LIN {X 0,Y 285.465,Z 322.576,A -85,B 0,C 180,E1 -17783.068,E2 -17783.068} C_VEL
LIN {X 0,Y 282.314,Z 318.057,A -85,B 0,C 180,E1 -17784.11,E2 -17784.11} C_VEL
LIN {X 0,Y 278.782,Z 313.124,A -85,B 0,C 180,E1 -17785.334,E2 -17785.334} C_VEL
LIN {X 0,Y 276.453,Z 310.274,A -85,B 0,C 180,E1 -17786.162,E2 -17786.162} C_VEL
LIN {X 0,Y 273.867,Z 306.493,A -85,B 0,C 180,E1 -17787.148,E2 -17787.148} C_VEL
LIN {X 0,Y 271.533,Z 304.482,A -85,B 0,C 180,E1 -17788.009,E2 -17788.009} C_VEL
LIN {X 0,Y 270.388,Z 302.092,A -85,B 0,C 180,E1 -17788.515,E2 -17788.515} C_VEL
LIN {X 0,Y 270.184,Z 301.141,A -85,B 0,C 180,E1 -17788.729,E2 -17788.729} C_VEL
LIN {X 0,Y 270.263,Z 301.128,A -85,B 0,C 180,E1 -17792.146,E2 -17792.146} C_VEL
LIN {X 0,Y 270.276,Z 301.125,A -85,B 0,C 180,E1 -17795.519,E2 -17795.519} C_VEL
LIN {X 0,Y 270.3,Z 301.092,A -85,B 0,C 180,E1 -17800.245,E2 -17800.245} C_VEL
LIN {X 0,Y 270.395,Z 301.089,A -85,B 0,C 180,E1 -17804.935,E2 -17804.935} C_VEL
LIN {X 0,Y 270.411,Z 301.113,A -85,B 0,C 180,E1 -17809.518,E2 -17809.518} C_VEL
LIN {X 0,Y 270.597,Z 301.053,A -85,B 0,C 180,E1 -17812.539,E2 -17812.539} C_VEL
LIN {X 0,Y 270.785,Z 301.051,A -85,B 0,C 180,E1 -17818.513,E2 -17818.513} C_VEL
LIN {X 0,Y 270.785,Z 301.026,A -85,B 0,C 180,E1 -17821.487,E2 -17821.487} C_VEL
LIN {X 0,Y 270.598,Z 301.049,A -85,B 0,C 180,E1 -17827.462,E2 -17827.462} C_VEL
LIN {X 0,Y 270.412,Z 301.097,A -85,B 0,C 180,E1 -17830.482,E2 -17830.482} C_VEL
LIN {X 0,Y 270.395,Z 301.076,A -85,B 0,C 180,E1 -17835.065,E2 -17835.065} C_VEL
LIN {X 0,Y 270.301,Z 301.113,A -85,B 0,C 180,E1 -17839.756,E2 -17839.756} C_VEL
LIN {X 0,Y 270.237,Z 301.135,A -85,B 0,C 180,E1 -17844.589,E2 -17844.589} C_VEL
LIN {X 0,Y 270.269,Z 301.1,A -85,B 0,C 180,E1 -17847.909,E2 -17847.909} C_VEL
LIN {X 0,Y 270.21,Z 301.225,A -85,B 0,C 180,E1 -17851.837,E2 -17851.837} C_VEL
LIN {X 0,Y 271.001,Z 303.633,A -85,B 0,C 180,E1 -17852.226,E2 -17852.226} C_VEL
LIN {X 0,Y 272.866,Z 305.851,A -85,B 0,C 180,E1 -17852.953,E2 -17852.953} C_VEL
LIN {X 0,Y 274.387,Z 306.942,A -85,B 0,C 180,E1 -17853.495,E2 -17853.495} C_VEL
LIN {X 0,Y 276.319,Z 310.113,A -85,B 0,C 180,E1 -17854.245,E2 -17854.245} C_VEL
LIN {X 0,Y 278.572,Z 312.374,A -85,B 0,C 180,E1 -17855.026,E2 -17855.026} C_VEL
LIN {X 0,Y 281.089,Z 315.815,A -85,B 0,C 180,E1 -17855.906,E2 -17855.906} C_VEL
LIN {X 0,Y 282.525,Z 317.531,A -85,B 0,C 180,E1 -17856.382,E2 -17856.382} C_VEL
LIN {X 0,Y 286.709,Z 323.191,A -85,B 0,C 180,E1 -17857.74,E2 -17857.74} C_VEL
LIN {X 0,Y 292.941,Z 331.669,A -85,B 0,C 180,E1 -17859.622,E2 -17859.622} C_VEL
LIN {X 0,Y 302.502,Z 345.885,A -85,B 0,C 180,E1 -17862.274,E2 -17862.274} C_VEL
LIN {X 0,Y 311.081,Z 359.947,A -85,B 0,C 180,E1 -17864.456,E2 -17864.456} C_VEL
LIN {X 0,Y 315.606,Z 368.338,A -85,B 0,C 180,E1 -17865.557,E2 -17865.557} C_VEL
LIN {X 0,Y 316.791,Z 370.757,A -85,B 0,C 180,E1 -17865.844,E2 -17865.844} C_VEL
LIN {X 0,Y 310.561,Z 496.144,A -85,B 0,C 180,E1 -17868.67,E2 -17868.67} C_VEL
LIN {X 0,Y 309.023,Z 512.229,A -85,B 0,C 180,E1 -17869.222,E2 -17869.222} C_VEL
LIN {X 0,Y 306.924,Z 528.349,A -85,B 0,C 180,E1 -17870.016,E2 -17870.016} C_VEL
LIN {X 0,Y 304.344,Z 543.648,A -85,B 0,C 180,E1 -17871.004,E2 -17871.004} C_VEL
LIN {X 0,Y 301.641,Z 556.838,A -85,B 0,C 180,E1 -17872.083,E2 -17872.083} C_VEL
LIN {X 0,Y 298.42,Z 570.73,A -85,B 0,C 180,E1 -17873.468,E2 -17873.468} C_VEL
LIN {X 0,Y 294.824,Z 584.321,A -85,B 0,C 180,E1 -17875.103,E2 -17875.103} C_VEL
LIN {X 0,Y 290.92,Z 597.703,A -85,B 0,C 180,E1 -17877.075,E2 -17877.075} C_VEL
LIN {X 0,Y 287.332,Z 609.078,A -85,B 0,C 180,E1 -17879.093,E2 -17879.093} C_VEL
LIN {X 0,Y 283.57,Z 620.478,A -85,B 0,C 180,E1 -17881.505,E2 -17881.505} C_VEL
LIN {X 0,Y 280.116,Z 630.242,A -85,B 0,C 180,E1 -17883.956,E2 -17883.956} C_VEL
LIN {X 0,Y 276.958,Z 639.603,A -85,B 0,C 180,E1 -17886.839,E2 -17886.839} C_VEL
LIN {X 0,Y 274.201,Z 647.442,A -85,B 0,C 180,E1 -17889.756,E2 -17889.756} C_VEL
LIN {X 0,Y 271.973,Z 654.426,A -85,B 0,C 180,E1 -17892.962,E2 -17892.962} C_VEL
LIN {X 0,Y 270.165,Z 660.416,A -85,B 0,C 180,E1 -17896.46,E2 -17896.46} C_VEL
LIN {X 0,Y 269.193,Z 664.308,A -85,B 0,C 180,E1 -17899.47,E2 -17899.47} C_VEL
LIN {X 0,Y 268.617,Z 667.199,A -85,B 0,C 180,E1 -17902.483,E2 -17902.483} C_VEL
LIN {X 0,Y 268.309,Z 669.097,A -85,B 0,C 180,E1 -17905.493,E2 -17905.493} C_VEL
LIN {X 0,Y 268.22,Z 670.055,A -85,B 0,C 180,E1 -17908.498,E2 -17908.498} C_VEL
LIN {X 0,Y 268.22,Z 670.068,A -85,B 0,C 180,E1 -17911.501,E2 -17911.501} C_VEL
LIN {X 0,Y 268.309,Z 669.159,A -85,B 0,C 180,E1 -17914.507,E2 -17914.507} C_VEL
LIN {X 0,Y 268.616,Z 667.287,A -85,B 0,C 180,E1 -17917.517,E2 -17917.517} C_VEL
LIN {X 0,Y 269.181,Z 664.444,A -85,B 0,C 180,E1 -17920.531,E2 -17920.531} C_VEL
LIN {X 0,Y 270.143,Z 660.575,A -85,B 0,C 180,E1 -17923.541,E2 -17923.541} C_VEL
LIN {X 0,Y 271.644,Z 655.594,A -85,B 0,C 180,E1 -17926.534,E2 -17926.534} C_VEL
LIN {X 0,Y 273.604,Z 649.5,A -85,B 0,C 180,E1 -17929.507,E2 -17929.507} C_VEL
LIN {X 0,Y 276.542,Z 641.01,A -85,B 0,C 180,E1 -17932.803,E2 -17932.803} C_VEL
LIN {X 0,Y 279.598,Z 631.844,A -85,B 0,C 180,E1 -17935.696,E2 -17935.696} C_VEL
LIN {X 0,Y 282.931,Z 622.4,A -85,B 0,C 180,E1 -17938.161,E2 -17938.161} C_VEL
LIN {X 0,Y 286.683,Z 611.383,A -85,B 0,C 180,E1 -17940.576,E2 -17940.576} C_VEL
LIN {X 0,Y 290.809,Z 598.342,A -85,B 0,C 180,E1 -17942.94,E2 -17942.94} C_VEL
LIN {X 0,Y 294.404,Z 586.186,A -85,B 0,C 180,E1 -17944.746,E2 -17944.746} C_VEL
LIN {X 0,Y 298.139,Z 572.182,A -85,B 0,C 180,E1 -17946.483,E2 -17946.483} C_VEL
LIN {X 0,Y 301.13,Z 559.648,A -85,B 0,C 180,E1 -17947.78,E2 -17947.78} C_VEL
LIN {X 0,Y 304.214,Z 544.829,A -85,B 0,C 180,E1 -17949.015,E2 -17949.015} C_VEL
LIN {X 0,Y 306.775,Z 529.881,A -85,B 0,C 180,E1 -17950.007,E2 -17950.007} C_VEL
LIN {X 0,Y 308.771,Z 515.295,A -85,B 0,C 180,E1 -17950.765,E2 -17950.765} C_VEL
LIN {X 0,Y 310.47,Z 498.633,A -85,B 0,C 180,E1 -17951.374,E2 -17951.374} C_VEL
LIN {X 0,Y 312.66,Z 454.995,A -85,B 0,C 180,E1 -17952.403,E2 -17952.403} C_VEL
LIN {X 0,Y 316.844,Z 370.753,A -85,B 0,C 180,E1 -17954.276,E2 -17954.276} C_VEL
LIN {X 0,Y 315.834,Z 368.672,A -85,B 0,C 180,E1 -17954.521,E2 -17954.521} C_VEL
LIN {X 0,Y 313.117,Z 364.696,A -85,B 0,C 180,E1 -17955.142,E2 -17955.142} C_VEL
LIN {X 0,Y 307.493,Z 359.894,A -85,B 0,C 180,E1 -17956.372,E2 -17956.372} C_VEL
LIN {X 0,Y 301.876,Z 355.264,A -85,B 0,C 180,E1 -17957.67,E2 -17957.67} C_VEL
LIN {X 0,Y 299.137,Z 351.53,A -85,B 0,C 180,E1 -17958.385,E2 -17958.385} C_VEL
LIN {X 0,Y 290.135,Z 337.942,A -85,B 0,C 180,E1 -17960.964,E2 -17960.964} C_VEL
LIN {X 0,Y 282.347,Z 327.012,A -85,B 0,C 180,E1 -17963.427,E2 -17963.427} C_VEL
LIN {X 0,Y 278.368,Z 321.874,A -85,B 0,C 180,E1 -17964.778,E2 -17964.778} C_VEL
LIN {X 0,Y 274.984,Z 317.484,A -85,B 0,C 180,E1 -17965.998,E2 -17965.998} C_VEL
LIN {X 0,Y 272.367,Z 314.328,A -85,B 0,C 180,E1 -17966.979,E2 -17966.979} C_VEL
LIN {X 0,Y 271.362,Z 312.806,A -85,B 0,C 180,E1 -17967.383,E2 -17967.383} C_VEL
LIN {X 0,Y 268.733,Z 310.164,A -85,B 0,C 180,E1 -17968.408,E2 -17968.408} C_VEL
LIN {X 0,Y 267.435,Z 307.674,A -85,B 0,C 180,E1 -17968.994,E2 -17968.994} C_VEL
LIN {X 0,Y 264.933,Z 305.894,A -85,B 0,C 180,E1 -17970.008,E2 -17970.008} C_VEL
LIN {X 0,Y 263.477,Z 303.347,A -85,B 0,C 180,E1 -17970.705,E2 -17970.705} C_VEL
LIN {X 0,Y 263.178,Z 301.998,A -85,B 0,C 180,E1 -17970.942,E2 -17970.942} C_VEL
LIN {X 0,Y 263.225,Z 302.01,A -85,B 0,C 180,E1 -17975.2,E2 -17975.2} C_VEL
LIN {X 0,Y 263.262,Z 301.988,A -85,B 0,C 180,E1 -17979.693,E2 -17979.693} C_VEL
LIN {X 0,Y 263.343,Z 301.96,A -85,B 0,C 180,E1 -17984.521,E2 -17984.521} C_VEL
LIN {X 0,Y 263.372,Z 301.961,A -85,B 0,C 180,E1 -17989.234,E2 -17989.234} C_VEL
LIN {X 0,Y 263.571,Z 301.946,A -85,B 0,C 180,E1 -17992.338,E2 -17992.338} C_VEL
LIN {X 0,Y 263.749,Z 301.914,A -85,B 0,C 180,E1 -17998.473,E2 -17998.473} C_VEL
LIN {X 0,Y 263.75,Z 301.935,A -85,B 0,C 180,E1 -18001.527,E2 -18001.527} C_VEL
LIN {X 0,Y 263.571,Z 301.966,A -85,B 0,C 180,E1 -18007.661,E2 -18007.661} C_VEL
LIN {X 0,Y 263.372,Z 301.956,A -85,B 0,C 180,E1 -18010.765,E2 -18010.765} C_VEL
LIN {X 0,Y 263.349,Z 301.987,A -85,B 0,C 180,E1 -18015.478,E2 -18015.478} C_VEL
LIN {X 0,Y 263.262,Z 302.006,A -85,B 0,C 180,E1 -18020.306,E2 -18020.306} C_VEL
LIN {X 0,Y 263.207,Z 302.012,A -85,B 0,C 180,E1 -18025.291,E2 -18025.291} C_VEL
LIN {X 0,Y 263.178,Z 302.022,A -85,B 0,C 180,E1 -18028.729,E2 -18028.729} C_VEL
LIN {X 0,Y 263.966,Z 304.47,A -85,B 0,C 180,E1 -18029.18,E2 -18029.18} C_VEL
LIN {X 0,Y 265.903,Z 306.766,A -85,B 0,C 180,E1 -18030.035,E2 -18030.035} C_VEL
LIN {X 0,Y 267.583,Z 308.046,A -85,B 0,C 180,E1 -18030.712,E2 -18030.712} C_VEL
LIN {X 0,Y 269.406,Z 311.041,A -85,B 0,C 180,E1 -18031.503,E2 -18031.503} C_VEL
LIN {X 0,Y 271.844,Z 313.447,A -85,B 0,C 180,E1 -18032.442,E2 -18032.442} C_VEL
LIN {X 0,Y 274.372,Z 316.935,A -85,B 0,C 180,E1 -18033.42,E2 -18033.42} C_VEL
LIN {X 0,Y 277.847,Z 321.57,A -85,B 0,C 180,E1 -18034.689,E2 -18034.689} C_VEL
LIN {X 0,Y 281.453,Z 326.899,A -85,B 0,C 180,E1 -18035.955,E2 -18035.955} C_VEL
LIN {X 0,Y 285.879,Z 333.543,A -85,B 0,C 180,E1 -18037.422,E2 -18037.422} C_VEL
LIN {X 0,Y 292.568,Z 344.244,A -85,B 0,C 180,E1 -18039.496,E2 -18039.496} C_VEL
LIN {X 0,Y 300.604,Z 358.33,A -85,B 0,C 180,E1 -18041.803,E2 -18041.803} C_VEL
LIN {X 0,Y 307.889,Z 372.775,A -85,B 0,C 180,E1 -18043.766,E2 -18043.766} C_VEL
LIN {X 0,Y 311.44,Z 380.362,A -85,B 0,C 180,E1 -18044.683,E2 -18044.683} C_VEL
LIN {X 0,Y 308.136,Z 444.749,A -85,B 0,C 180,E1 -18046.131,E2 -18046.131} C_VEL
LIN {X 0,Y 304.665,Z 511.319,A -85,B 0,C 180,E1 -18047.67,E2 -18047.67} C_VEL
LIN {X 0,Y 302.695,Z 528.883,A -85,B 0,C 180,E1 -18048.292,E2 -18048.292} C_VEL
LIN {X 0,Y 300.31,Z 544.128,A -85,B 0,C 180,E1 -18049.06,E2 -18049.06} C_VEL
LIN {X 0,Y 297.723,Z 557.974,A -85,B 0,C 180,E1 -18049.965,E2 -18049.965} C_VEL
LIN {X 0,Y 294.414,Z 572.93,A -85,B 0,C 180,E1 -18051.199,E2 -18051.199} C_VEL
LIN {X 0,Y 290.49,Z 588.182,A -85,B 0,C 180,E1 -18052.783,E2 -18052.783} C_VEL
LIN {X 0,Y 286.436,Z 602.162,A -85,B 0,C 180,E1 -18054.573,E2 -18054.573} C_VEL
LIN {X 0,Y 282.601,Z 614.107,A -85,B 0,C 180,E1 -18056.404,E2 -18056.404} C_VEL
LIN {X 0,Y 278.871,Z 625.337,A -85,B 0,C 180,E1 -18058.471,E2 -18058.471} C_VEL
LIN {X 0,Y 275.078,Z 636.542,A -85,B 0,C 180,E1 -18060.959,E2 -18060.959} C_VEL
LIN {X 0,Y 271.178,Z 647.403,A -85,B 0,C 180,E1 -18063.859,E2 -18063.859} C_VEL
LIN {X 0,Y 268.007,Z 656.542,A -85,B 0,C 180,E1 -18066.837,E2 -18066.837} C_VEL
LIN {X 0,Y 265.507,Z 664.21,A -85,B 0,C 180,E1 -18069.873,E2 -18069.873} C_VEL
LIN {X 0,Y 263.315,Z 671.784,A -85,B 0,C 180,E1 -18073.652,E2 -18073.652} C_VEL
LIN {X 0,Y 261.866,Z 677.78,A -85,B 0,C 180,E1 -18077.602,E2 -18077.602} C_VEL
LIN {X 0,Y 261.237,Z 681.216,A -85,B 0,C 180,E1 -18080.711,E2 -18080.711} C_VEL
LIN {X 0,Y 261.034,Z 683.72,A -85,B 0,C 180,E1 -18083.818,E2 -18083.818} C_VEL
LIN {X 0,Y 261.048,Z 685.135,A -85,B 0,C 180,E1 -18086.914,E2 -18086.914} C_VEL
LIN {X 0,Y 261.125,Z 685.667,A -85,B 0,C 180,E1 -18090,E2 -18090} C_VEL
LIN {X 0,Y 261.048,Z 685.126,A -85,B 0,C 180,E1 -18093.087,E2 -18093.087} C_VEL
LIN {X 0,Y 261.034,Z 683.701,A -85,B 0,C 180,E1 -18096.182,E2 -18096.182} C_VEL
LIN {X 0,Y 261.237,Z 681.189,A -85,B 0,C 180,E1 -18099.289,E2 -18099.289} C_VEL
LIN {X 0,Y 261.865,Z 677.744,A -85,B 0,C 180,E1 -18102.398,E2 -18102.398} C_VEL
LIN {X 0,Y 263.311,Z 671.738,A -85,B 0,C 180,E1 -18106.346,E2 -18106.346} C_VEL
LIN {X 0,Y 265.511,Z 664.142,A -85,B 0,C 180,E1 -18110.127,E2 -18110.127} C_VEL
LIN {X 0,Y 268.478,Z 655.196,A -85,B 0,C 180,E1 -18113.624,E2 -18113.624} C_VEL
LIN {X 0,Y 272.105,Z 644.819,A -85,B 0,C 180,E1 -18116.872,E2 -18116.872} C_VEL
LIN {X 0,Y 275.954,Z 633.851,A -85,B 0,C 180,E1 -18119.658,E2 -18119.658} C_VEL
LIN {X 0,Y 279.474,Z 623.397,A -85,B 0,C 180,E1 -18121.876,E2 -18121.876} C_VEL
LIN {X 0,Y 283.551,Z 610.848,A -85,B 0,C 180,E1 -18124.109,E2 -18124.109} C_VEL
LIN {X 0,Y 287.49,Z 598.427,A -85,B 0,C 180,E1 -18125.923,E2 -18125.923} C_VEL
LIN {X 0,Y 291.256,Z 585.073,A -85,B 0,C 180,E1 -18127.537,E2 -18127.537} C_VEL
LIN {X 0,Y 294.847,Z 570.849,A -85,B 0,C 180,E1 -18128.952,E2 -18128.952} C_VEL
LIN {X 0,Y 298.179,Z 555.513,A -85,B 0,C 180,E1 -18130.182,E2 -18130.182} C_VEL
LIN {X 0,Y 300.955,Z 539.768,A -85,B 0,C 180,E1 -18131.166,E2 -18131.166} C_VEL
LIN {X 0,Y 303.256,Z 523.658,A -85,B 0,C 180,E1 -18131.892,E2 -18131.892} C_VEL
LIN {X 0,Y 304.847,Z 507.548,A -85,B 0,C 180,E1 -18132.401,E2 -18132.401} C_VEL
LIN {X 0,Y 311.342,Z 380.373,A -85,B 0,C 180,E1 -18135.293,E2 -18135.293} C_VEL
LIN {X 0,Y 303.557,Z 364.081,A -85,B 0,C 180,E1 -18137.338,E2 -18137.338} C_VEL
LIN {X 0,Y 295.854,Z 349.879,A -85,B 0,C 180,E1 -18139.484,E2 -18139.484} C_VEL
LIN {X 0,Y 288.564,Z 337.824,A -85,B 0,C 180,E1 -18141.663,E2 -18141.663} C_VEL
LIN {X 0,Y 282.355,Z 328.23,A -85,B 0,C 180,E1 -18143.671,E2 -18143.671} C_VEL
LIN {X 0,Y 276.499,Z 319.625,A -85,B 0,C 180,E1 -18145.726,E2 -18145.726} C_VEL
LIN {X 0,Y 271.891,Z 313.543,A -85,B 0,C 180,E1 -18147.454,E2 -18147.454} C_VEL
LIN {X 0,Y 271.042,Z 312.597,A -85,B 0,C 180,E1 -18147.78,E2 -18147.78} C_VEL
LIN {X 0,Y 268.535,Z 309.887,A -85,B 0,C 180,E1 -18148.767,E2 -18148.767} C_VEL
LIN {X 0,Y 267.428,Z 307.691,A -85,B 0,C 180,E1 -18149.269,E2 -18149.269} C_VEL
LIN {X 0,Y 264.827,Z 305.742,A -85,B 0,C 180,E1 -18150.324,E2 -18150.324} C_VEL
LIN {X 0,Y 263.543,Z 303.548,A -85,B 0,C 180,E1 -18150.932,E2 -18150.932} C_VEL
LIN {X 0,Y 263.193,Z 302.012,A -85,B 0,C 180,E1 -18151.163,E2 -18151.163} C_VEL
LIN {X 0,Y 263.225,Z 302.003,A -85,B 0,C 180,E1 -18155.2,E2 -18155.2} C_VEL
LIN {X 0,Y 263.262,Z 301.968,A -85,B 0,C 180,E1 -18159.694,E2 -18159.694} C_VEL
LIN {X 0,Y 263.343,Z 301.973,A -85,B 0,C 180,E1 -18164.522,E2 -18164.522} C_VEL
LIN {X 0,Y 263.354,Z 301.988,A -85,B 0,C 180,E1 -18169.234,E2 -18169.234} C_VEL
LIN {X 0,Y 263.557,Z 301.931,A -85,B 0,C 180,E1 -18172.338,E2 -18172.338} C_VEL
LIN {X 0,Y 263.75,Z 301.927,A -85,B 0,C 180,E1 -18178.473,E2 -18178.473} C_VEL
LIN {X 0,Y 263.749,Z 301.901,A -85,B 0,C 180,E1 -18181.527,E2 -18181.527} C_VEL
LIN {X 0,Y 263.557,Z 301.924,A -85,B 0,C 180,E1 -18187.662,E2 -18187.662} C_VEL
LIN {X 0,Y 263.354,Z 301.982,A -85,B 0,C 180,E1 -18190.767,E2 -18190.767} C_VEL
LIN {X 0,Y 263.344,Z 301.953,A -85,B 0,C 180,E1 -18195.479,E2 -18195.479} C_VEL
LIN {X 0,Y 263.262,Z 301.979,A -85,B 0,C 180,E1 -18200.307,E2 -18200.307} C_VEL
LIN {X 0,Y 263.192,Z 302.013,A -85,B 0,C 180,E1 -18205.293,E2 -18205.293} C_VEL
LIN {X 0,Y 263.162,Z 301.994,A -85,B 0,C 180,E1 -18209.279,E2 -18209.279} C_VEL
LIN {X 0,Y 263.946,Z 304.503,A -85,B 0,C 180,E1 -18209.731,E2 -18209.731} C_VEL
LIN {X 0,Y 265.82,Z 306.72,A -85,B 0,C 180,E1 -18210.553,E2 -18210.553} C_VEL
LIN {X 0,Y 267.578,Z 308.003,A -85,B 0,C 180,E1 -18211.256,E2 -18211.256} C_VEL
LIN {X 0,Y 269.417,Z 311.056,A -85,B 0,C 180,E1 -18212.052,E2 -18212.052} C_VEL
LIN {X 0,Y 271.859,Z 313.427,A -85,B 0,C 180,E1 -18212.985,E2 -18212.985} C_VEL
LIN {X 0,Y 274.324,Z 316.869,A -85,B 0,C 180,E1 -18213.937,E2 -18213.937} C_VEL
LIN {X 0,Y 275.947,Z 318.646,A -85,B 0,C 180,E1 -18214.519,E2 -18214.519} C_VEL
LIN {X 0,Y 278.959,Z 322.471,A -85,B 0,C 180,E1 -18215.583,E2 -18215.583} C_VEL
LIN {X 0,Y 286.344,Z 332.572,A -85,B 0,C 180,E1 -18218.022,E2 -18218.022} C_VEL
LIN {X 0,Y 294.128,Z 343.854,A -85,B 0,C 180,E1 -18220.357,E2 -18220.357} C_VEL
LIN {X 0,Y 301.981,Z 356.159,A -85,B 0,C 180,E1 -18222.522,E2 -18222.522} C_VEL
LIN {X 0,Y 309.792,Z 369.68,A -85,B 0,C 180,E1 -18224.528,E2 -18224.528} C_VEL
LIN {X 0,Y 311.653,Z 373.831,A -85,B 0,C 180,E1 -18225.011,E2 -18225.011} C_VEL
LIN {X 0,Y 305.247,Z 496.823,A -85,B 0,C 180,E1 -18227.803,E2 -18227.803} C_VEL
LIN {X 0,Y 303.576,Z 513.363,A -85,B 0,C 180,E1 -18228.384,E2 -18228.384} C_VEL
LIN {X 0,Y 301.51,Z 528.565,A -85,B 0,C 180,E1 -18229.148,E2 -18229.148} C_VEL
LIN {X 0,Y 298.863,Z 543.862,A -85,B 0,C 180,E1 -18230.148,E2 -18230.148} C_VEL
LIN {X 0,Y 296.053,Z 557.052,A -85,B 0,C 180,E1 -18231.236,E2 -18231.236} C_VEL
LIN {X 0,Y 292.661,Z 571.225,A -85,B 0,C 180,E1 -18232.671,E2 -18232.671} C_VEL
LIN {X 0,Y 289.008,Z 584.533,A -85,B 0,C 180,E1 -18234.294,E2 -18234.294} C_VEL
LIN {X 0,Y 284.948,Z 597.915,A -85,B 0,C 180,E1 -18236.293,E2 -18236.293} C_VEL
LIN {X 0,Y 281.203,Z 609.29,A -85,B 0,C 180,E1 -18238.342,E2 -18238.342} C_VEL
LIN {X 0,Y 277.301,Z 620.689,A -85,B 0,C 180,E1 -18240.799,E2 -18240.799} C_VEL
LIN {X 0,Y 273.712,Z 630.453,A -85,B 0,C 180,E1 -18243.299,E2 -18243.299} C_VEL
LIN {X 0,Y 270.382,Z 639.814,A -85,B 0,C 180,E1 -18246.241,E2 -18246.241} C_VEL
LIN {X 0,Y 267.498,Z 647.652,A -85,B 0,C 180,E1 -18249.226,E2 -18249.226} C_VEL
LIN {X 0,Y 265.033,Z 654.942,A -85,B 0,C 180,E1 -18252.675,E2 -18252.675} C_VEL
LIN {X 0,Y 263.24,Z 660.625,A -85,B 0,C 180,E1 -18256.097,E2 -18256.097} C_VEL
LIN {X 0,Y 262.187,Z 664.517,A -85,B 0,C 180,E1 -18259.185,E2 -18259.185} C_VEL
LIN {X 0,Y 261.553,Z 667.408,A -85,B 0,C 180,E1 -18262.279,E2 -18262.279} C_VEL
LIN {X 0,Y 261.223,Z 669.305,A -85,B 0,C 180,E1 -18265.37,E2 -18265.37} C_VEL
LIN {X 0,Y 261.148,Z 670.262,A -85,B 0,C 180,E1 -18268.458,E2 -18268.458} C_VEL
LIN {X 0,Y 261.148,Z 670.274,A -85,B 0,C 180,E1 -18271.542,E2 -18271.542} C_VEL
LIN {X 0,Y 261.223,Z 669.367,A -85,B 0,C 180,E1 -18274.629,E2 -18274.629} C_VEL
LIN {X 0,Y 261.551,Z 667.495,A -85,B 0,C 180,E1 -18277.721,E2 -18277.721} C_VEL
LIN {X 0,Y 262.174,Z 664.652,A -85,B 0,C 180,E1 -18280.815,E2 -18280.815} C_VEL
LIN {X 0,Y 263.213,Z 660.783,A -85,B 0,C 180,E1 -18283.904,E2 -18283.904} C_VEL
LIN {X 0,Y 264.969,Z 655.241,A -85,B 0,C 180,E1 -18287.281,E2 -18287.281} C_VEL
LIN {X 0,Y 267.441,Z 647.924,A -85,B 0,C 180,E1 -18290.779,E2 -18290.779} C_VEL
LIN {X 0,Y 270.349,Z 640.148,A -85,B 0,C 180,E1 -18293.762,E2 -18293.762} C_VEL
LIN {X 0,Y 273.649,Z 630.829,A -85,B 0,C 180,E1 -18296.708,E2 -18296.708} C_VEL
LIN {X 0,Y 277.702,Z 619.658,A -85,B 0,C 180,E1 -18299.571,E2 -18299.571} C_VEL
LIN {X 0,Y 281.501,Z 608.588,A -85,B 0,C 180,E1 -18301.913,E2 -18301.913} C_VEL
LIN {X 0,Y 285.829,Z 595.359,A -85,B 0,C 180,E1 -18304.225,E2 -18304.225} C_VEL
LIN {X 0,Y 289.36,Z 584.041,A -85,B 0,C 180,E1 -18305.87,E2 -18305.87} C_VEL
LIN {X 0,Y 292.881,Z 570.526,A -85,B 0,C 180,E1 -18307.53,E2 -18307.53} C_VEL
LIN {X 0,Y 296.329,Z 556.334,A -85,B 0,C 180,E1 -18308.939,E2 -18308.939} C_VEL
LIN {X 0,Y 299.351,Z 541.909,A -85,B 0,C 180,E1 -18310.102,E2 -18310.102} C_VEL
LIN {X 0,Y 301.915,Z 526.191,A -85,B 0,C 180,E1 -18311.117,E2 -18311.117} C_VEL
LIN {X 0,Y 304.074,Z 510.004,A -85,B 0,C 180,E1 -18311.865,E2 -18311.865} C_VEL
LIN {X 0,Y 305.508,Z 493.753,A -85,B 0,C 180,E1 -18312.396,E2 -18312.396} C_VEL
LIN {X 0,Y 311.684,Z 374.516,A -85,B 0,C 180,E1 -18315.094,E2 -18315.094} C_VEL
LIN {X 0,Y 311.524,Z 373.054,A -85,B 0,C 180,E1 -18315.17,E2 -18315.17} C_VEL
LIN {X 0,Y 306.539,Z 363.74,A -85,B 0,C 180,E1 -18316.432,E2 -18316.432} C_VEL
LIN {X 0,Y 299.137,Z 351.53,A -85,B 0,C 180,E1 -18318.385,E2 -18318.385} C_VEL
LIN {X 0,Y 297.216,Z 349.296,A -85,B 0,C 180,E1 -18318.888,E2 -18318.888} C_VEL
LIN {X 0,Y 293.211,Z 347.423,A -85,B 0,C 180,E1 -18319.868,E2 -18319.868} C_VEL
LIN {X 0,Y 289.153,Z 345.776,A -85,B 0,C 180,E1 -18320.902,E2 -18320.902} C_VEL
LIN {X 0,Y 287.132,Z 343.847,A -85,B 0,C 180,E1 -18321.48,E2 -18321.48} C_VEL
LIN {X 0,Y 279.278,Z 332.662,A -85,B 0,C 180,E1 -18324.045,E2 -18324.045} C_VEL
LIN {X 0,Y 275.302,Z 327.48,A -85,B 0,C 180,E1 -18325.444,E2 -18325.444} C_VEL
LIN {X 0,Y 272.245,Z 323.49,A -85,B 0,C 180,E1 -18326.584,E2 -18326.584} C_VEL
LIN {X 0,Y 269.355,Z 319.721,A -85,B 0,C 180,E1 -18327.719,E2 -18327.719} C_VEL
LIN {X 0,Y 265.752,Z 315.503,A -85,B 0,C 180,E1 -18329.198,E2 -18329.198} C_VEL
LIN {X 0,Y 264.941,Z 314.011,A -85,B 0,C 180,E1 -18329.575,E2 -18329.575} C_VEL
LIN {X 0,Y 262.36,Z 311.786,A -85,B 0,C 180,E1 -18330.678,E2 -18330.678} C_VEL
LIN {X 0,Y 260.414,Z 308.524,A -85,B 0,C 180,E1 -18331.641,E2 -18331.641} C_VEL
LIN {X 0,Y 257.85,Z 306.666,A -85,B 0,C 180,E1 -18332.836,E2 -18332.836} C_VEL
LIN {X 0,Y 256.522,Z 304.414,A -85,B 0,C 180,E1 -18333.563,E2 -18333.563} C_VEL
LIN {X 0,Y 256.135,Z 302.875,A -85,B 0,C 180,E1 -18333.849,E2 -18333.849} C_VEL
LIN {X 0,Y 256.098,Z 302.866,A -85,B 0,C 180,E1 -18337.406,E2 -18337.406} C_VEL
LIN {X 0,Y 256.186,Z 302.887,A -85,B 0,C 180,E1 -18340.78,E2 -18340.78} C_VEL
LIN {X 0,Y 256.278,Z 302.838,A -85,B 0,C 180,E1 -18344.083,E2 -18344.083} C_VEL
LIN {X 0,Y 256.293,Z 302.873,A -85,B 0,C 180,E1 -18347.328,E2 -18347.328} C_VEL
LIN {X 0,Y 256.479,Z 302.811,A -85,B 0,C 180,E1 -18350.56,E2 -18350.56} C_VEL
LIN {X 0,Y 256.486,Z 302.85,A -85,B 0,C 180,E1 -18353.707,E2 -18353.707} C_VEL
LIN {X 0,Y 256.712,Z 302.789,A -85,B 0,C 180,E1 -18358.431,E2 -18358.431} C_VEL
LIN {X 0,Y 256.713,Z 302.809,A -85,B 0,C 180,E1 -18361.569,E2 -18361.569} C_VEL
LIN {X 0,Y 256.538,Z 302.839,A -85,B 0,C 180,E1 -18367.873,E2 -18367.873} C_VEL
LIN {X 0,Y 256.308,Z 302.836,A -85,B 0,C 180,E1 -18371.066,E2 -18371.066} C_VEL
LIN {X 0,Y 256.298,Z 302.867,A -85,B 0,C 180,E1 -18375.915,E2 -18375.915} C_VEL
LIN {X 0,Y 256.165,Z 302.885,A -85,B 0,C 180,E1 -18380.895,E2 -18380.895} C_VEL
LIN {X 0,Y 256.159,Z 302.892,A -85,B 0,C 180,E1 -18385.501,E2 -18385.501} C_VEL
LIN {X 0,Y 256.182,Z 303.104,A -85,B 0,C 180,E1 -18385.834,E2 -18385.834} C_VEL
LIN {X 0,Y 256.962,Z 305.457,A -85,B 0,C 180,E1 -18386.333,E2 -18386.333} C_VEL
LIN {X 0,Y 259.006,Z 307.755,A -85,B 0,C 180,E1 -18387.36,E2 -18387.36} C_VEL
LIN {X 0,Y 260.738,Z 308.888,A -85,B 0,C 180,E1 -18388.146,E2 -18388.146} C_VEL
LIN {X 0,Y 262.518,Z 311.96,A -85,B 0,C 180,E1 -18389.027,E2 -18389.027} C_VEL
LIN {X 0,Y 265.188,Z 314.537,A -85,B 0,C 180,E1 -18390.179,E2 -18390.179} C_VEL
LIN {X 0,Y 267.566,Z 317.889,A -85,B 0,C 180,E1 -18391.207,E2 -18391.207} C_VEL
LIN {X 0,Y 269.314,Z 319.694,A -85,B 0,C 180,E1 -18391.9,E2 -18391.9} C_VEL
LIN {X 0,Y 274.902,Z 327.279,A -85,B 0,C 180,E1 -18394.059,E2 -18394.059} C_VEL
LIN {X 0,Y 281.991,Z 337.92,A -85,B 0,C 180,E1 -18396.567,E2 -18396.567} C_VEL
LIN {X 0,Y 289.58,Z 350.372,A -85,B 0,C 180,E1 -18399.014,E2 -18399.014} C_VEL
LIN {X 0,Y 297.365,Z 364.377,A -85,B 0,C 180,E1 -18401.321,E2 -18401.321} C_VEL
LIN {X 0,Y 304.245,Z 378.418,A -85,B 0,C 180,E1 -18403.239,E2 -18403.239} C_VEL
LIN {X 0,Y 306.421,Z 383.051,A -85,B 0,C 180,E1 -18403.821,E2 -18403.821} C_VEL
LIN {X 0,Y 299.483,Z 510.885,A -85,B 0,C 180,E1 -18406.75,E2 -18406.75} C_VEL
LIN {X 0,Y 297.534,Z 527.769,A -85,B 0,C 180,E1 -18407.342,E2 -18407.342} C_VEL
LIN {X 0,Y 294.974,Z 543.929,A -85,B 0,C 180,E1 -18408.155,E2 -18408.155} C_VEL
LIN {X 0,Y 291.889,Z 559.763,A -85,B 0,C 180,E1 -18409.224,E2 -18409.224} C_VEL
LIN {X 0,Y 288.476,Z 574.383,A -85,B 0,C 180,E1 -18410.471,E2 -18410.471} C_VEL
LIN {X 0,Y 284.546,Z 589.02,A -85,B 0,C 180,E1 -18412.032,E2 -18412.032} C_VEL
LIN {X 0,Y 280.256,Z 603.134,A -85,B 0,C 180,E1 -18413.892,E2 -18413.892} C_VEL
LIN {X 0,Y 276.64,Z 613.9,A -85,B 0,C 180,E1 -18415.58,E2 -18415.58} C_VEL
LIN {X 0,Y 272.778,Z 625.13,A -85,B 0,C 180,E1 -18417.683,E2 -18417.683} C_VEL
LIN {X 0,Y 268.827,Z 636.335,A -85,B 0,C 180,E1 -18420.217,E2 -18420.217} C_VEL
LIN {X 0,Y 265.195,Z 645.953,A -85,B 0,C 180,E1 -18422.797,E2 -18422.797} C_VEL
LIN {X 0,Y 261.588,Z 655.736,A -85,B 0,C 180,E1 -18425.988,E2 -18425.988} C_VEL
LIN {X 0,Y 258.741,Z 664,A -85,B 0,C 180,E1 -18429.323,E2 -18429.323} C_VEL
LIN {X 0,Y 256.324,Z 671.834,A -85,B 0,C 180,E1 -18433.35,E2 -18433.35} C_VEL
LIN {X 0,Y 254.85,Z 677.571,A -85,B 0,C 180,E1 -18437.255,E2 -18437.255} C_VEL
LIN {X 0,Y 254.181,Z 681.008,A -85,B 0,C 180,E1 -18440.451,E2 -18440.451} C_VEL
LIN {X 0,Y 253.944,Z 683.512,A -85,B 0,C 180,E1 -18443.644,E2 -18443.644} C_VEL
LIN {X 0,Y 253.948,Z 684.928,A -85,B 0,C 180,E1 -18446.827,E2 -18446.827} C_VEL
LIN {X 0,Y 254.052,Z 685.461,A -85,B 0,C 180,E1 -18450,E2 -18450} C_VEL
LIN {X 0,Y 253.948,Z 684.918,A -85,B 0,C 180,E1 -18453.173,E2 -18453.173} C_VEL
LIN {X 0,Y 253.944,Z 683.493,A -85,B 0,C 180,E1 -18456.356,E2 -18456.356} C_VEL
LIN {X 0,Y 254.181,Z 680.98,A -85,B 0,C 180,E1 -18459.549,E2 -18459.549} C_VEL
LIN {X 0,Y 255.099,Z 676.452,A -85,B 0,C 180,E1 -18463.543,E2 -18463.543} C_VEL
LIN {X 0,Y 256.323,Z 671.787,A -85,B 0,C 180,E1 -18466.65,E2 -18466.65} C_VEL
LIN {X 0,Y 258.195,Z 665.588,A -85,B 0,C 180,E1 -18469.892,E2 -18469.892} C_VEL
LIN {X 0,Y 260.696,Z 658.288,A -85,B 0,C 180,E1 -18473.01,E2 -18473.01} C_VEL
LIN {X 0,Y 263.837,Z 649.578,A -85,B 0,C 180,E1 -18476.073,E2 -18476.073} C_VEL
LIN {X 0,Y 267.783,Z 639.163,A -85,B 0,C 180,E1 -18479.047,E2 -18479.047} C_VEL
LIN {X 0,Y 270.985,Z 629.996,A -85,B 0,C 180,E1 -18481.245,E2 -18481.245} C_VEL
LIN {X 0,Y 275.297,Z 617.653,A -85,B 0,C 180,E1 -18483.728,E2 -18483.728} C_VEL
LIN {X 0,Y 279.451,Z 605.263,A -85,B 0,C 180,E1 -18485.783,E2 -18485.783} C_VEL
LIN {X 0,Y 283.886,Z 590.926,A -85,B 0,C 180,E1 -18487.713,E2 -18487.713} C_VEL
LIN {X 0,Y 287.621,Z 577.27,A -85,B 0,C 180,E1 -18489.216,E2 -18489.216} C_VEL
LIN {X 0,Y 291.461,Z 561.39,A -85,B 0,C 180,E1 -18490.62,E2 -18490.62} C_VEL
LIN {X 0,Y 294.512,Z 546.063,A -85,B 0,C 180,E1 -18491.696,E2 -18491.696} C_VEL
LIN {X 0,Y 297.202,Z 529.796,A -85,B 0,C 180,E1 -18492.544,E2 -18492.544} C_VEL
LIN {X 0,Y 299.197,Z 513.228,A -85,B 0,C 180,E1 -18493.144,E2 -18493.144} C_VEL
LIN {X 0,Y 300.657,Z 488.11,A -85,B 0,C 180,E1 -18493.785,E2 -18493.785} C_VEL
LIN {X 0,Y 306.301,Z 382.981,A -85,B 0,C 180,E1 -18496.16,E2 -18496.16} C_VEL
LIN {X 0,Y 298.575,Z 366.821,A -85,B 0,C 180,E1 -18498.281,E2 -18498.281} C_VEL
LIN {X 0,Y 291.561,Z 353.961,A -85,B 0,C 180,E1 -18500.319,E2 -18500.319} C_VEL
